// ---- XTS/Mover/types/ST_GEAR_DATA.TcDUT
{attribute 'pack_mode' := '2'}
TYPE ST_GEAR_DATA :
STRUCT
  rDeltaToMasterPos       : LREAL := 100.0;
  rModuloSyncPosSlave     : LREAL := 225.0;
  rMasterStartDistance    : LREAL :=   0.0;
  rGearNumerator          : LREAL :=   1.0;
  iGearDenumerator        : USINT :=   1;
END_STRUCT
END_TYPE

// ---- XTS/XtsStation/_types/ST_STATION_PARAMETER.TcDUT
TYPE ST_STATION_PARAMETER :
STRUCT
  sText             : STRING(80); // only description
  rPosWait          : REAL;       // start of station, a sending station is using this value to send mover to
  rReleaseDistance  : REAL;       // distance mover has to travel (from ActPos) in order for station to go back to mover detection

  rGap              : REAL;
  rVelo             : REAL;
  rAccDec           : REAL;
  rJerk             : REAL;

  // how many nests (stop positions) mover has to stop at (1 = default)
  nConfiguredStopCount  : USINT := 1; // 1-8 --> NestMask = BYTE

  // mover stop position in station, relative to rPosWait!!
  rPosStop          : ARRAY[1..8] OF LREAL;
END_STRUCT
END_TYPE

// ---- XTS/Xpu/types/ST_XPU_CTRL.TcDUT
{attribute 'pack_mode' := '2'}
TYPE ST_XPU_CTRL :
STRUCT
  Cmd             : E_XPU_CTRL;
END_STRUCT
END_TYPE

// ---- APPLICATION/GVL_APPLICATION.TcGVL
VAR_GLOBAL CONSTANT
  MAX_PROCESS       : UINT := 3;
END_VAR
{attribute 'qualified_only'}
VAR_GLOBAL
  MasterAxis              : Tc2_MC2.AXIS_REF;

  MasterPower             : Tc2_MC2.MC_Power;
  MasterReset             : Tc2_MC2.MC_Reset;
  MasterHalt              : Tc2_MC2.MC_Halt;
  MasterMoveVelo          : Tc2_MC2.MC_MoveVelocity;

  MoveData                : ST_MOVE_DATA;    // dynamic constraints for move commands
  GearData                : ST_GEAR_DATA;    // dynamic constraints and positions for GearIn/GearInPosCa

END_VAR

// ---- MSG/GVL_MSG.TcGVL
{attribute 'qualified_only'}
VAR_GLOBAL CONSTANT
  //-----------------------------------------------------------------------------
  // file paths for message system
  //  - compiler define option WIN switches to Windows file paths
  //-----------------------------------------------------------------------------
{IF defined (WIN)}
  {info 'WIN folders'}
  LOG_DIR               : STRING  := 'C:\TwinCAT\#MsgFiles\';
  CONFIG_DIR            : STRING  := 'C:\TwinCAT\XPU_PLC_StationConfig\';
{ELSE}
  {info 'BSD folders'}
  LOG_DIR               : STRING  := '/usr/local/etc/TwinCAT/#MsgFiles/';
  CONFIG_DIR            : STRING  := '/usr/local/etc/TwinCAT/XPU_PLC_StationConfig/';
{END_IF}

  LOG_FILE              : STRING  := 'MSG_XtsTransport_';
  CONFIG_FILE           : STRING  := 'Config_XPU_'; // OTCID of fb_Environment is added to name on writing

  MAX_MESSAGE           : UINT    := 200; // max entry in message list
END_VAR
VAR_GLOBAL
  Messages                        : ARRAY[1..MAX_MESSAGE] OF ST_Message;
  MessageIndex                    : UINT := 0; // message index
  MessageError                    : UINT := 0; // error counter

  fbLocalTime                     : fb_LocalTime;
  dtLocalTime                     : DT;
  sLocalTime                      : STRING;

  MessageLevelXpu                 : E_MessageType;
  MessageLevelStations            : ARRAY[1..MAX_STATION] OF E_MessageType;
  MessageLevelMovers              : ARRAY[1..MAX_MOVER]   OF E_MessageType;

  MessageLevelProcess             : ARRAY[1..MAX_PROCESS] OF E_MessageType;

{IF defined (TEST)}
  {info 'TEST logging enabled'}
  MessageLevel                    : E_MessageType := eMessageVerbose; // a lot of messages
{ELSE}
  MessageLevel                    : E_MessageType := eMessageError;    // not as much messages 
{END_IF}

END_VAR

// ---- XTS/GVL_XTS.TcGVL
{attribute 'qualified_only'}
VAR_GLOBAL
  //---------------------------------------------------------------------------
  // XTS Station
  //  - handshakes mover in station with extern control
  //  - station parameters (positions, gap, dyn. constraints, description...)
  StationStart        : ST_STATION_PARAMETER;   // Xts transport is sending all mover to this position (CMD_TRANSPORT_START)
  StationStartIndex   : UINT := 1;              // index of XtsStation where all movers are entered into linked list.

  // station handshaking with mover and extern process
  // station sends mover to target station/WaitPos
  // station adds mover data to LinkedList.AddTail() of target station
  Station             : ARRAY[1..MAX_STATION] OF fb_Station;
  StationList         : ARRAY[1..MAX_STATION] OF fb_Station_LinkedListCtrl;

  StationQueue        : ARRAY[1..MAX_STATION]    OF 
                        ARRAY[1..MAX_LIST_NODES] OF ST_STATION_MOVER_DATA;

  // interface for access to List methods
  StationListItf      : ARRAY[1..MAX_STATION] OF I_Station_LinkedList;

  // interface for access to station methods
  StationCtrlItf      : ARRAY[1..MAX_STATION] OF I_XtsTransport_Station;

  // ctrl / state datafields for extern control
  StationCtrl         : ARRAY[1..MAX_STATION] OF ST_STATION_CTRL;   // control for extern to write
  StationState        : ARRAY[1..MAX_STATION] OF ST_STATION_STATE;  // state for extern to read

  // station parameter
  StationParameter    : ARRAY[1..MAX_STATION] OF ST_STATION_PARAMETER; // XtsStation (fb_Station) positions and dyn constraints

  // static position offsets in stations
  PositionOffset      : ARRAY[1..MAX_STATION] OF T_NEST_OFFSET; // added to PosStop[] in XtsStation


  //---------------------------------------------------------------------------
  // XTS
  // XTS TransportUnit
  //  - handles request for XPU, Group, Mover, StartUp, ReStart
  XtsTransport        : fb_TransportUnit;         // manages members of XTS transport for extern to access

  XtsTransportCtrl    : ST_XTS_TRANSPORT_CTRL;    // control of XTS transport for extern to write
  XtsTransportState   : ST_XTS_TRANSPORT_STATE;   // state   of XTS transport for extern to read


  //---------------------------------------------------------------------------
  // XPU
  // XTS-Utility checks
  // XTS-Utility interfaces for you to use
  Xpu             : fb_XpuCtrl;

  XpuCtrl         : ST_XPU_CTRL;
  XpuState        : ST_XPU_STATE;
  XpuInfo         : ST_XPU_INFO;
  XpuModules      : ARRAY[1..MAX_MODULE] OF Tc3_XTS_Utility.ST_InfoDataView;


  //---------------------------------------------------------------------------
  // Collision avoidance group CA
  //
  // - add mover to group
  // - build group
  // - clear group
  CaGroup         : FB_CaGroup;                   // cyclic check of CaGroup state and errors; carries methods for handling CaGroup
  CaGroupItf      : I_XtsTransport_CaGroup;       // Interface used by fb_TransportUnit

  // cyclic mapping to MOTION/Objects/CaGroup 
  CaGroupRef      : Tc3_McCoordinatedMotion.AXES_GROUP_REF;

  // Info data from CaGroup FB
  CaGroupInfo     : ST_GROUP_INFO;                // cyclic info about CaGroup for fb_TransportUnit to read
  //---------------------------------------------------------------------------

  //---------------------------------------------------------------------------
  // MC2 encapsulation, CA movement
  Mover           : ARRAY[1..MAX_MOVER] OF fb_MoverCtrl;    // MC and CA methods for mover; cyclic check for individual command on mover

  MoverCtrl       : ARRAY[1..MAX_MOVER] OF ST_MOVER_CTRL;   // control of individual mover for extern to write
  MoverState      : ARRAY[1..MAX_MOVER] OF ST_MOVER_STATE;  // state   of individual mover for extern to read

  MoverItf        : ARRAY[1..MAX_MOVER] OF I_XtsTransport_Mover;  // Interface used by fb_TransportUnit

  LastPosition    : ARRAY[1..MAX_MOVER] OF LREAL;           // on execute of any movement, value is saved here (used by fb_Mover)
  LastGap         : ARRAY[1..MAX_MOVER] OF LREAL;           // on execute of any movement, value is saved here (used by fb_Mover)

  MoverInfo       : ARRAY[1..MAX_MOVER] OF ST_MOVER_INFO;   // cyclic info about mover for extern to read

  MoveData        : ARRAY[1..MAX_MOVER] OF ST_MOVE_DATA;    // dynamic constraints for move commands
  GearData        : ARRAY[1..MAX_MOVER] OF ST_GEAR_DATA;    // dynamic constraints and positions for GearIn/GearInPosCa
  
  // cyclic mapping to MOTION/Axes
  AxisRefMover    : ARRAY[1..MAX_MOVER] OF Tc2_MC2.AXIS_REF;
  //---------------------------------------------------------------------------
END_VAR

// ---- XTS/XTS_Parameter.TcGVL
//{attribute 'qualified_only'}
VAR_GLOBAL CONSTANT
// HAUD 2025 08 09
//
//    XTS_TRANSPORT_LAYER project
//    
//    MIT License
//    
//    Copyright (c) 2025 HAUD
//    
//    Permission is hereby granted, free of charge, to any person obtaining a copy
//    of this software and associated documentation files (the "Software"), to deal
//    in the Software without restriction, including without limitation the rights
//    to use, copy, modify, merge, publish, distribute, sublicense, and/or sell
//    copies of the Software, and to permit persons to whom the Software is
//    furnished to do so, subject to the following conditions:
//    
//    The above copyright notice and this permission notice shall be included in all
//    copies or substantial portions of the Software.
//    
//    THE SOFTWARE IS PROVIDED "AS IS", WITHOUT WARRANTY OF ANY KIND, EXPRESS OR
//    IMPLIED, INCLUDING BUT NOT LIMITED TO THE WARRANTIES OF MERCHANTABILITY,
//    FITNESS FOR A PARTICULAR PURPOSE AND NONINFRINGEMENT. IN NO EVENT SHALL THE
//    AUTHORS OR COPYRIGHT HOLDERS BE LIABLE FOR ANY CLAIM, DAMAGES OR OTHER
//    LIABILITY, WHETHER IN AN ACTION OF CONTRACT, TORT OR OTHERWISE, ARISING FROM,
//    OUT OF OR IN CONNECTION WITH THE SOFTWARE OR THE USE OR OTHER DEALINGS IN THE
//    SOFTWARE.

  Version             : STRING  := '4.00.11';

  MAX_MOVER           : UINT    := TO_UINT(Tc3_XTS_Utility.TcIoXtsEnvironmentParameterList.MaxXtsMoversPerXpu);
  MAX_MODULE          : UINT    := TO_UINT(Tc3_XTS_Utility.TcIoXtsEnvironmentParameterList.MaxModulesPerPart);
  MAX_PART            : UINT    := TO_UINT(Tc3_XTS_Utility.TcIoXtsEnvironmentParameterList.MaxXtsPartsPerXpu);
  MAX_TRACK           : UINT    := TO_UINT(Tc3_XTS_Utility.TcIoXtsEnvironmentParameterList.MaxXtsTracksPerXpu);
  MAX_GROUP           : UINT    := TO_UINT(Tc3_XTS_Utility.TcIoXtsEnvironmentParameterList.MaxXtsCaGroup);

  MAX_INFO_SERVER     : UINT    := TO_UINT(Tc3_XTS_Utility.TcIoXtsEnvironmentParameterList.MaxXtsInfoServer);
  MAX_INFO_STATION    : UINT    := TO_UINT(Tc3_XTS_Utility.TcIoXtsEnvironmentParameterList.MaxXtsInfoStation);
  MAX_INFO_STOP_POS   : UINT    := TO_UINT(Tc3_XTS_Utility.TcIoXtsEnvironmentParameterList.MaxXtsStopPositionsPerStation);

  MAX_PARAMETER_SET   : UINT    := TO_UINT(Tc3_XTS_Utility.TcIoXtsEnvironmentParameterList.MaxXtsParameterSet);

  MAX_NCT_BASE_UNIT   : UINT    := TO_UINT(Tc3_XTS_Utility.TcIoXtsEnvironmentParameterList.MaxXtsNctBaseUnitInterfaces);

  MAX_STATION         : UINT    := 2;

  MAX_STATION_NEST    : UINT    := TO_UINT(SIZEOF(ST_STATION_STATE.nMask)*8);
  // MAX_LIST_NODES      : UINT    := MAX_MOVER;
  MAX_LIST_NODES      : UINT    := 24; // visualization can not handle access to MAX_MOVER
  MAX_MASTER          : UINT    := 1;
END_VAR

// ---- XTS/Mover/I_XtsTransport_Mover.TcIO
INTERFACE I_XtsTransport_Mover

METHOD Disable : E_PROGRESS
VAR_INPUT
  Execute             : BOOL;
END_VAR
END_METHOD

METHOD Enable : E_PROGRESS
VAR_INPUT
  Execute             : BOOL;
END_VAR
END_METHOD

METHOD GearIn : E_PROGRESS;
VAR_INPUT
  Execute             : BOOL;
  stMoveData          : ST_MOVE_DATA;
  stGearData          : ST_GEAR_DATA;
END_VAR
END_METHOD

METHOD GearInPosCa : E_PROGRESS
VAR_INPUT
  Execute             : BOOL;
  stMoveData          : ST_MOVE_DATA;
  stGearData          : ST_GEAR_DATA;  
END_VAR
END_METHOD

METHOD GearOut : E_PROGRESS
VAR_INPUT
  Execute             : BOOL;
END_VAR
END_METHOD

METHOD Halt : E_PROGRESS
VAR_INPUT
  Execute             : BOOL;
  stMoveData          : ST_MOVE_DATA;
END_VAR
END_METHOD

METHOD HaltCa : E_PROGRESS
VAR_INPUT
  Execute             : BOOL;
  stMoveData          : ST_MOVE_DATA;
END_VAR
END_METHOD

PROPERTY MessageLevel : e_messagetype
SET
END_SET
END_PROPERTY

PROPERTY ModuloTurn : dint
GET
END_GET
END_PROPERTY

METHOD MoveToPos : E_PROGRESS
VAR_INPUT
  Execute             : BOOL;
  stMoveData          : ST_MOVE_DATA;
END_VAR
END_METHOD

METHOD MoveToPosCa : E_PROGRESS
VAR_INPUT
  Execute             : BOOL;
  stMoveData          : ST_MOVE_DATA;
END_VAR
END_METHOD

PROPERTY RailLength : LREAL
GET
END_GET
SET
END_SET
END_PROPERTY

METHOD Reset : E_PROGRESS
VAR_INPUT
  Execute             : BOOL;
END_VAR
END_METHOD

METHOD SendToAbsPosCa : E_PROGRESS
VAR_INPUT
  Execute             : BOOL;
  stMoveData          : ST_MOVE_DATA;
END_VAR
END_METHOD

METHOD SendToModuloPosCa : E_PROGRESS
VAR_INPUT
  Execute             : BOOL;
  stMoveData          : ST_MOVE_DATA;
END_VAR
END_METHOD

METHOD Stop : E_PROGRESS
VAR_INPUT
  Execute             : BOOL;
  stMoveData          : ST_MOVE_DATA;
END_VAR
END_METHOD

END_INTERFACE

// ---- MAIN.TcPOU
//---------------------------------------------------------------------------------------------------------------
//
//  HAUD 2024.10.02
//
//  - XTS_DEMO_GEAR_IN_POS_CA
//
//  - XTS_TRANSPORT_LAYER
//  - transport layer members:
//    - CaGroup
//      - access to Group functions
//
//    - Mover
//      - access to MC and CA motion functions
//
//    - Xpu (ProcessingUnit)
//      - access to TcCOM Objects in Environment
//
//    - Transport Control Unit
//      - coordinates members to get XTS in defined states
//
//  - global datafields for mrmbers in GVL_XTS namespace
//  - global interface datafields for use in members
//  - structures are assigned by reference for every member
//
//---------------------------------------------------------------------------------------------------------------
// HAUD 2024 05 29
//
//    XTS_TRANSPORT_LAYER project
//    
//    MIT License
//    
//    Copyright (c) 2024 HAUD
//    
//    Permission is hereby granted, free of charge, to any person obtaining a copy
//    of this software and associated documentation files (the "Software"), to deal
//    in the Software without restriction, including without limitation the rights
//    to use, copy, modify, merge, publish, distribute, sublicense, and/or sell
//    copies of the Software, and to permit persons to whom the Software is
//    furnished to do so, subject to the following conditions:
//    
//    The above copyright notice and this permission notice shall be included in all
//    copies or substantial portions of the Software.
//    
//    THE SOFTWARE IS PROVIDED "AS IS", WITHOUT WARRANTY OF ANY KIND, EXPRESS OR
//    IMPLIED, INCLUDING BUT NOT LIMITED TO THE WARRANTIES OF MERCHANTABILITY,
//    FITNESS FOR A PARTICULAR PURPOSE AND NONINFRINGEMENT. IN NO EVENT SHALL THE
//    AUTHORS OR COPYRIGHT HOLDERS BE LIABLE FOR ANY CLAIM, DAMAGES OR OTHER
//    LIABILITY, WHETHER IN AN ACTION OF CONTRACT, TORT OR OTHERWISE, ARISING FROM,
//    OUT OF OR IN CONNECTION WITH THE SOFTWARE OR THE USE OR OTHER DEALINGS IN THE
//    SOFTWARE.
//---------------------------------------------------------------------------------------------------------------
PROGRAM MAIN
VAR
	bInit 				: BOOL;
  eInit         : E_PROGRESS;

  nStation,
	nMover,
  nMoverSelected,
  nStationSelected,
  nStationParameter   : UINT;

  sStationText        : STRING(30);

  eTransportState     : E_XTS_TRANSPORT_STATE;
  eTransportResult    : E_PROGRESS;

  eXpuState           : E_XPU_STATE;
  eXpuResult          : E_PROGRESS;
  eXpuCheck           : E_XPU_CHECK;

  eMoverState         : E_MOVER_STATE;
  eMoverResult        : E_PROGRESS;

  sCaGroupState,
  sTransportState,
  sTransportCheck,
  sTransportResult,
  sXpuState,
  sXpuResult,
  sXpuCheck,
  sXpuOpMode,
  sXpuMoverdetectionMode,
  sXpuMoverAssignement,
  sMoverState,
  sMoverResult,
  sStationState,
  sStationStateMask,
  sStationCtrlMask        : STRING;

  bStationEnable,
  bStationEnter,
  bStationStart,
  bStationDone,
  bStationOut,
  bStationGone            : BOOL;

  tStationSelectedQueue   : ARRAY[1..MAX_LIST_NODES] OF ST_STATION_MOVER_DATA;

  tonWriteLog             : Tc2_Standard.TON;
  tWriteLog               : TIME := T#5S;
END_VAR

//############################################################################
// Local time; used for timestamps
//############################################################################
GVL_MSG.fbLocalTime(
                    sLocalTime                => GVL_MSG.sLocalTime, 
                    dtLocalTime               => GVL_MSG.dtLocalTime);
//############################################################################

//############################################################################
// 	example for init sequence
//############################################################################	
IF NOT bInit
THEN
  CASE eInit
  OF
    E_PROGRESS.PROGRESS_INVALID,
    E_PROGRESS.PROGRESS_DONE:         // clear command interface
      eInit                                   := E_PROGRESS.PROGRESS_BUSY;
      GVL_XTS.XpuCtrl.Cmd                     := E_XPU_CTRL.XTS_CMD_NULL;
      GVL_MSG.MessageLevelXpu                 := GVL_MSG.MessageLevel;
      GVL_XTS.CaGroup.MessageLevel            := GVL_MSG.MessageLevel;
      FOR nStation := 1 TO MAX_STATION
      DO
        GVL_MSG.MessageLevelStations[nStation]:= GVL_MSG.MessageLevel;
      END_FOR
      FOR nMover := 1 TO MAX_MOVER
      DO
        GVL_MSG.MessageLevelMovers[nMover]    := GVL_MSG.MessageLevel;
      END_FOR


    E_PROGRESS.PROGRESS_BUSY:         // init Xpu, ProcessingUnit, MotorModules
      eInit                                   := E_PROGRESS.PROGRESS_PREPARE;
      GVL_XTS.XpuCtrl.Cmd                     := E_XPU_CTRL.XTS_CMD_INIT;

    E_PROGRESS.PROGRESS_PREPARE:      // wait for init to be done
      IF (GVL_XTS.XpuState.State      = E_XPU_STATE.XTS_INIT + E_PROGRESS.PROGRESS_DONE)
      THEN
        eInit                                 := E_PROGRESS.PROGRESS_STARTUP;
        GVL_XTS.XpuCtrl.Cmd                   := E_XPU_CTRL.XTS_IDLE;
      END_IF

    E_PROGRESS.PROGRESS_STARTUP:      // assign mover interfaces
      eInit                                   := E_PROGRESS.PROGRESS_CHECK;
      FOR nMover := 1 TO MAX_MOVER
      DO
        GVL_XTS.MoverItf[nMover]              := GVL_XTS.Mover[nMover];
      END_FOR

    E_PROGRESS.PROGRESS_CHECK:        // assign CaGroup interface
      eInit                                   := E_PROGRESS.PROGRESS_OCCUPIED;
      GVL_XTS.CaGroupItf                      := GVL_XTS.CaGroup;

    E_PROGRESS.PROGRESS_OCCUPIED:     // StartStation for XtsTransportCtrl.Cmd := E_XTS_TRANSPORT_CTRL.CMD_TRANSPORT_START;
      eInit                                   := E_PROGRESS.PROGRESS_WORKING;
      // where to start?
      GVL_XTS.XtsTransport.StationStartIndex  := 0; // no stations in use in this example, therefore no StartStation

      // IF you use stations, initialize them here, before StationStart is initialized!

    E_PROGRESS.PROGRESS_WORKING:
      // Start Position parameters
      GVL_XTS.StationStart.rPosWait           :=     10.0; // this value may differ from the GVL_XTS.StationParameter[StartStationIndex], IF it differs, you MUST have room for positive movement to GVL_XTS.StationParameter[StartStationIndex].rWaitPos
      GVL_XTS.StationStart.rGap               :=    250.0; // may differ, or just copy from GVL_XTS.StationParameter[StartStationIndex]
      GVL_XTS.StationStart.rVelo              :=    750.0; // may differ, or just copy from GVL_XTS.StationParameter[StartStationIndex]
      GVL_XTS.StationStart.rAccDec            :=  12000.0; // may differ, or just copy from GVL_XTS.StationParameter[StartStationIndex]
      GVL_XTS.StationStart.rJerk              := 400000.0; // may differ, or just copy from GVL_XTS.StationParameter[StartStationIndex], the movements are more robust if you keep this value in a narrow range, since jumps lead to adjusting movements within the CA Group

      IF (GVL_XTS.XtsTransport.StationStartIndex > 0) AND
         (GVL_XTS.XtsTransport.StationStartIndex < MAX_STATION+1)
      THEN
        GVL_XTS.StationStart.nConfiguredStopCount := GVL_XTS.StationParameter[GVL_XTS.XtsTransport.StationStartIndex].nConfiguredStopCount;
      END_IF

      bInit                                           := TRUE;
      eInit                                           := E_PROGRESS.PROGRESS_DONE;
  END_CASE
END_IF

//############################################################################
// 	XTS Transport Unit
//############################################################################
//  - main control function block for transport layer
//  - requires access to member controls
//    - Xpu
//    - CaGroup
//    - Mover
//    - Station Control
//    - Station LinkedList Interface
//############################################################################
//
// cyclic call
GVL_XTS.XtsTransport();

// main control
GVL_XTS.XtsTransport.Ctrl               REF= GVL_XTS.XtsTransportCtrl;   // main control
GVL_XTS.XtsTransport.State              REF= GVL_XTS.XtsTransportState;  // main state
                                        
// member controls                      
GVL_XTS.XtsTransport.XpuCtrl            REF= GVL_XTS.XpuCtrl;
GVL_XTS.XtsTransport.XpuState           REF= GVL_XTS.XpuState;
GVL_XTS.XtsTransport.XpuInfo            REF= GVL_XTS.XpuInfo;
                                        
GVL_XTS.XtsTransport.GroupItf           :=   GVL_XTS.CaGroupItf;
GVL_XTS.XtsTransport.GroupInfo          REF= GVL_XTS.CaGroupInfo;
                                        
GVL_XTS.XtsTransport.MoverItf           REF= GVL_XTS.MoverItf;
GVL_XTS.XtsTransport.MoverInfo          REF= GVL_XTS.MoverInfo;
GVL_XTS.XtsTransport.MoverLastPosition  REF= GVL_XTS.LastPosition;
GVL_XTS.XtsTransport.MoverLastGap       REF= GVL_XTS.LastGap;
                                        
GVL_XTS.XtsTransport.StationStart       REF= GVL_XTS.StationStart;      // start position for E_XTS_TRANSPORT_CTRL.CMD_TRANSPORT_START
GVL_XTS.XtsTransport.StationCtrlItf     REF= GVL_XTS.StationCtrlItf;    // station interfaces are required for accessing station methods
GVL_XTS.XtsTransport.StationListsItf    REF= GVL_XTS.StationListItf;    // list interface is required for access to linked list methods
GVL_XTS.XtsTransport.StationControl     REF= GVL_XTS.StationCtrl;
GVL_XTS.XtsTransport.StationState       REF= GVL_XTS.StationState;
//############################################################################



//############################################################################
// 	XTS Stations
//############################################################################	
FOR nStation := 1 TO MAX_STATION
DO
  GVL_XTS.Station[nStation].StationId   := nStation;
  GVL_XTS.Station[nStation].MessageLevel:= GVL_MSG.MessageLevelStations[nStation];

  GVL_XTS.StationListItf[nStation]      := GVL_XTS.StationList[nStation];   // interfaces for list methods
  GVL_XTS.StationCtrlItf[nStation]      := GVL_XTS.Station[nStation];       // interfaces for station methods

  GVL_XTS.Station[nStation].Ctrl        REF= GVL_XTS.StationCtrl;           // station ctrl from extern
  GVL_XTS.Station[nStation].State       REF= GVL_XTS.StationState;          // station state to extern

  GVL_XTS.Station[nStation].ItfStations REF= GVL_XTS.StationListItf;        // give every station all list interfaces for writing mover tickets
  GVL_XTS.Station[nStation].ItfMover    REF= GVL_XTS.MoverItf;              // give every station all mover interfaces for movement in / out of station
  GVL_XTS.Station[nStation].Mover       REF= GVL_XTS.AxisRefMover;          // AXIS_REF to read infos from
  GVL_XTS.Station[nStation].MoverOffset REF= GVL_XTS.PositionOffset;        // static offsets for all stations, all movers, all stop positions


  GVL_XTS.Station[nStation].StationParameter  REF= GVL_XTS.StationParameter;// give every station all station parameters for sending to WaitPos of target station

  // cyclic call
  GVL_XTS.Station[nStation].Cycle();                                        // cycle for handshaking with extern

  // Queue data for each station
  GVL_XTS.StationQueue[nStation]        := GVL_XTS.StationListItf[nStation].Data;
END_FOR
//############################################################################



//############################################################################
// 	XPU environment
//############################################################################	
GVL_XTS.Xpu.XpuInstance               :=   1;
GVL_XTS.Xpu.MessageLevel              :=   GVL_MSG.MessageLevelXpu;

GVL_XTS.Xpu.Ctrl                      REF= GVL_XTS.XpuCtrl;
GVL_XTS.Xpu.State                     REF= GVL_XTS.XpuState;
GVL_XTS.Xpu.XpuModuleInfoData         REF= GVL_XTS.XpuModules;

GVL_XTS.Xpu.CaGroupOID                :=   GVL_XTS.CaGroup.GroupInfo.CaGroupOID;

// cyclic call
GVL_XTS.Xpu();
GVL_XTS.XpuInfo                       :=   GVL_XTS.Xpu.XpuInfo;
//############################################################################


//############################################################################	
// 	CA-Group Class
//############################################################################	
// assignment
GVL_XTS.CaGroup.AxisRef               REF= GVL_XTS.AxisRefMover;
// Interface to Mover methods
GVL_XTS.CaGroup.MoverItf              REF= GVL_XTS.MoverItf; 

GVL_XTS.CaGroup.GroupRef              REF= GVL_XTS.CaGroupRef;

// cyclic call
GVL_XTS.CaGroup.InfoCycle(TRUE); // read group status

// InfoData from group
GVL_XTS.CaGroupInfo                   :=   GVL_XTS.CaGroup.GroupInfo;

// Interface of CaGroup
GVL_XTS.CaGroupItf                    :=   GVL_XTS.CaGroup;
//############################################################################


//############################################################################
// Mover Class	
//############################################################################	
FOR nMover := 1 TO MAX_MOVER
DO
  GVL_XTS.Mover[nMover].MoverId       :=   nMover;
  GVL_XTS.Mover[nMover].RailLength    :=   GVL_XTS.Xpu.RailLength;  // mover needs RailLength, in order to calc absolute position from modulo input
  GVL_XTS.Mover[nMover].MessageLevel  :=   GVL_MSG.MessageLevelMovers[nMover];

  GVL_XTS.Mover[nMover].Ctrl          REF= GVL_XTS.MoverCtrl;       // mover control from extern
  GVL_XTS.Mover[nMover].State         REF= GVL_XTS.MoverState;      // mover state to extern

  GVL_XTS.Mover[nMover].MoveData      REF= GVL_XTS.MoveData;        // dyn constraints for extern to write
  GVL_XTS.Mover[nMover].GearData      REF= GVL_XTS.GearData;        // GearIn/GearInPosCa data fro extern to write

  // assignment	
  GVL_XTS.Mover[nMover].Mover         REF= GVL_XTS.AxisRefMover[nMover];  // axis reference to Mover function block
  GVL_XTS.Mover[nMover].LastGap       REF= GVL_XTS.LastGap[nMover];       // reference to last used gap value datafield
  GVL_XTS.Mover[nMover].LastPosition  REF= GVL_XTS.LastPosition[nMover];  // reference to last position datafield

  GVL_XTS.Mover[nMover].MoverInfo		  REF= GVL_XTS.MoverInfo[nMover];     // refernence to mover info data (ActPos, SetPos, ...)

  GVL_XTS.MoverItf[nMover]            :=   GVL_XTS.Mover[nMover];

  // master axis assigned to mover
  GVL_XTS.Mover[nMover].Master        REF= GVL_APPLICATION.MasterAxis;    // GearInPosCa conveyer axis is master in this example

  // cyclic call
  GVL_XTS.Mover[nMover].Cycle();  // call AXIS_REF()
  GVL_XTS.Mover[nMover]();        // call Ctrl/State
END_FOR


//############################################################################


//############################################################################
// /logging
//############################################################################
tonWriteLog(IN:= TRUE, PT := tWriteLog);

IF (tonWriteLog.Q)
THEN
  MessageData.bWriteFile      := TRUE;
  tonWriteLog(IN:= FALSE);
END_IF

//-----------------------------------------------------------------------------------------------------------------
// write message list to file
//-----------------------------------------------------------------------------------------------------------------
MessageData(pList			        := ADR(GVL_MSG.Messages),
			      pLocalTime        := ADR(GVL_MSG.dtLocalTime), 
			      bBusy=> );

// clear write trigger
IF MessageData.bWriteFile AND
   MessageData.bDone
THEN
  MessageData.bWriteFile      := FALSE;
END_IF
//############################################################################
// logging/
//############################################################################



//############################################################################
// Visualization data	
//############################################################################	
// get enumerations from XPU for visu:
eTransportState                       := f_GetState   (GVL_XTS.XtsTransportState.State);
eTransportResult                      := f_GetProgress(GVL_XTS.XtsTransportState.State);

eXpuState                             := f_GetState   (GVL_XTS.XpuState.State);
eXpuResult                            := f_GetProgress(GVL_XTS.XpuState.State);

eXpuCheck                             := GVL_XTS.XpuState.Check;

// display xpu state and result in visu
// get strings and info
sCaGroupState                         := TO_STRING(GVL_XTS.CaGroupInfo.CaGroupState);

sTransportState                       := TO_STRING(eTransportState);
sTransportCheck                       := TO_STRING(GVL_XTS.XtsTransportState.Check);
sTransportResult                      := TO_STRING(eTransportResult);

sXpuState                             := TO_STRING(eXpuState);
sXpuResult                            := TO_STRING(eXpuResult);
sXpuCheck                             := TO_STRING(eXpuCheck);

sXpuOpMode                            := GVL_XTS.Xpu.OpModeToString();
sXpuMoverdetectionMode                := GVL_XTS.Xpu.IdDetectionModeToString();
sXpuMoverAssignement                  := GVL_XTS.Xpu.MoverPositionAssignementToString();

nMoverSelected                        := SEL((nMoverSelected<1), nMoverSelected, 1);
nMoverSelected                        := SEL((nMoverSelected>MAX_MOVER), nMoverSelected, MAX_MOVER);

nStationSelected                      := SEL((nStationSelected<1), nStationSelected, 1);
nStationSelected                      := SEL((nStationSelected>MAX_STATION), nStationSelected, MAX_STATION);

bStationEnable                        := SEL((GVL_XTS.StationCtrl[nStationSelected].eCmd = E_STATION_CTRL.STATION_ENABLE),        FALSE, TRUE);
bStationEnter                         := SEL((GVL_XTS.StationCtrl[nStationSelected].eCmd = E_STATION_CTRL.STATION_MOVER_ENTER),   FALSE, TRUE);
bStationStart                         := SEL((GVL_XTS.StationCtrl[nStationSelected].eCmd = E_STATION_CTRL.STATION_PROCESS_START), FALSE, TRUE);
bStationDone                          := SEL((GVL_XTS.StationCtrl[nStationSelected].eCmd = E_STATION_CTRL.STATION_PROCESS_DONE),  FALSE, TRUE);
bStationOut                           := SEL((GVL_XTS.StationCtrl[nStationSelected].eCmd = E_STATION_CTRL.STATION_MOVER_OUT),     FALSE, TRUE);
bStationGone                          := SEL((GVL_XTS.StationCtrl[nStationSelected].eCmd = E_STATION_CTRL.STATION_MOVER_GONE),    FALSE, TRUE);

eMoverState                           := f_GetState   (GVL_XTS.MoverState[nMoverSelected].State);
eMoverResult                          := f_GetProgress(GVL_XTS.MoverState[nMoverSelected].State);

sMoverState                           := TO_STRING(eMoverState);
sMoverResult                          := TO_STRING(eMoverResult);

sStationState                         := TO_STRING(GVL_XTS.StationState[nStationSelected].eState);
sStationStateMask                     := Tc2_Utilities.BYTE_TO_BINSTR(GVL_XTS.StationState[nStationSelected].nMask, 8);
sStationCtrlMask                      := Tc2_Utilities.BYTE_TO_BINSTR(GVL_XTS.StationCtrl[nStationSelected].nMask, 8);

tStationSelectedQueue                 := GVL_XTS.StationQueue[nStationSelected];

END_PROGRAM

// ---- MSG/MessageData.TcPOU
PROGRAM MessageData
VAR CONSTANT
{attribute 'hide'}
  STR_LEN       : UDINT := 131_070;
END_VAR
VAR_INPUT
	bPowerFail		: BOOL;   // UPS switch
	bWriteFile		: BOOL;   // manual write of list
	bReset				: BOOL;
	pList					: POINTER TO ARRAY[1..GVL_MSG.MAX_MESSAGE] OF ST_Message; // attach your list here
	pLocalTime		: POINTER TO DT; 
END_VAR
VAR_OUTPUT
	bBusy					: BOOL;
  bDone         : BOOL;
	VisuList		  : ARRAY[1..GVL_MSG.MAX_MESSAGE] OF ST_Message;
END_VAR
VAR
	eState 				: E_MESSAGE_STATE;

	rtrigReset		: Tc2_Standard.R_TRIG;
	aWriteList		: ARRAY[1..GVL_MSG.MAX_MESSAGE] OF ST_Message;
	sWriteData		: STRING(STR_LEN);
	sNewLine			: STRING := '$N';
	sTab					: STRING := '$T';
	iCount, 
	iStart, 
	iEnd					: UINT;

	fbCreateDir		: Tc2_System.FB_CreateDir;
	sTmp          : STRING(256);
	sFilename			: STRING(256);
	sFolderDate		: STRING;
	bFileCreated	: BOOL;

	fbFileOpen		  : Tc2_System.FB_FileOpen;
	fbFileWrite		  : Tc2_System.FB_FileWrite;
	fbFileClose		  : Tc2_System.FB_FileClose;

  ivis          : UINT;

  bBusyWrite,
  bErrorWrite   : BOOL;
  nErrorWrite   : UDINT;
  nStateWrite   : UINT;
END_VAR

//-----------------------------------------------------------------------------
// check pointers
//-----------------------------------------------------------------------------
IF NOT (pList <> 0) OR
   NOT (pLocalTime <> 0)
THEN
  eState                      := MSG_INVALID_POINTERS;
  RETURN;
END_IF
//-----------------------------------------------------------------------------
// check date
// new message file for a new day
//-----------------------------------------------------------------------------
IF (FolderDate(pLocalTime) <> sFolderDate)
THEN
  bFileCreated                := FALSE;
END_IF
//-----------------------------------------------------------------------------
//----------------------------------------------------------------------------- 
rtrigReset(CLK:= bReset);
IF rtrigReset.Q
THEN
  bReset                      := FALSE;
  eState                      := MSG_NULL;
END_IF
//-----------------------------------------------------------------------------
//-----------------------------------------------------------------------------
CASE eState OF
  MSG_NULL:
    bBusy                     := 
    bDone                     := FALSE;

    IF (GVL_MSG.MessageIndex > GVL_MSG.MAX_MESSAGE/2)
    THEN
      eState                  := MSG_INIT;

    ELSIF (bWriteFile) OR (bPowerFail)
    THEN
      eState                  := MSG_INIT;

      IF (GVL_MSG.MessageIndex = 0)
      THEN
        bBusy                 := TRUE;
        eState                := MSG_WRITE_FILE_DONE;
      END_IF
    END_IF
END_CASE
//-----------------------------------------------------------------------------
CASE eState OF
  MSG_INIT:
    WriteData(FALSE);

    // clear intern list
    memset(ADR(aWriteList),     0, SIZEOF(aWriteList));

    // copy from attached list to local
    memcpy(ADR(aWriteList), pList, SIZEOF(aWriteList));

    // clear attached list
    memset(pList, 0, SIZEOF(aWriteList));

    bBusy                     := TRUE;
    iStart 	                  := 1;
    iEnd 		                  := SEL((GVL_MSG.MessageIndex > GVL_MSG.MAX_MESSAGE-1),
                                      GVL_MSG.MessageIndex,
                                      GVL_MSG.MAX_MESSAGE);
    GVL_MSG.MessageIndex      := 0;

    IF NOT bFileCreated
    THEN
      // folder and filename have to be created
      eState                  := MSG_ROOT;
    ELSE
      // folder and file already exist
      eState                  := MSG_LINE_START;
    END_IF
END_CASE
//-----------------------------------------------------------------------------
CASE eState OF
  MSG_ROOT:
    eState                    := MSG_ROOT_CREATE;
    fbCreateDir.sPathName     := left(GVL_MSG.LOG_DIR,len(GVL_MSG.LOG_DIR)-1);
    fbCreateDir(
            bExecute	        := FALSE);
  
  MSG_ROOT_CREATE:
    (* create root folder *)
    fbCreateDir(
            bExecute	        := TRUE);
    IF fbCreateDir.bBusy
    THEN
      eState                  := MSG_ROOT_CREATE_BUSY;
    END_IF
  
  MSG_ROOT_CREATE_BUSY:
    fbCreateDir(
            bExecute	        := TRUE);
    IF NOT fbCreateDir.bBusy
    THEN
      eState                  := MSG_FOLDER;
    END_IF
  
  MSG_FOLDER:
    eState                    := MSG_FOLDER_CREATE;
    sFolderDate               := FolderDate(pLocalTime);
    fbCreateDir.sPathName     := concat(GVL_MSG.LOG_DIR, sFolderDate);
    fbCreateDir(
            bExecute	        := FALSE);

  MSG_FOLDER_CREATE:
    (* create active folder *)
    fbCreateDir(
            bExecute	        := TRUE);
    IF fbCreateDir.bBusy
    THEN
      eState                  := MSG_FOLDER_CREATE_BUSY;
    END_IF
  
  MSG_FOLDER_CREATE_BUSY:
    fbCreateDir(
            bExecute	        := TRUE);
    IF NOT fbCreateDir.bBusy
    THEN
      eState                  := MSG_FILE_CREATE_DONE;
      fbCreateDir(
              bExecute	      := FALSE);
    END_IF
END_CASE
//-----------------------------------------------------------------------------
CASE eState OF
  MSG_FILE_CREATE_DONE:
    eState                    := MSG_LINE_START;
    bFileCreated              := TRUE;
    // build complete file path
    sTmp                      := concat(concat(GVL_MSG.LOG_FILE, sFolderDate),'.txt');
    sTmp                      := concat('\', sTmp);
    sFilename                 := concat(fbCreateDir.sPathName, sTmp);
END_CASE
//-----------------------------------------------------------------------------
CASE eState OF
  MSG_LINE_START:
    GVL_MSG.MessageError      := 0;
    eState                    := MSG_LINE_BUILD;
    iCount                    := iStart;
    memset(ADR(sWriteData),0,SIZEOF(sWriteData));
END_CASE
//-----------------------------------------------------------------------------
CASE eState OF
  MSG_LINE_BUILD:
    eState                    := MSG_LINE_CHECK;
    IF (aWriteList[iCount].eType > E_MessageType.eMessageEmpty)
    THEN
      sTmp                    := TO_STRING(aWriteList[iCount].eType);
      sTmp                    := Tc2_Standard.CONCAT(sTmp, sTab);
      sTmp                    := Tc2_Standard.CONCAT(sTmp, aWriteList[iCount].tTime);
      sTmp                    := Tc2_Standard.CONCAT(sTmp, sTab);
      sTmp                    := Tc2_Standard.CONCAT(sTmp, Device_To_String(aWriteList[iCount].eDevice));
      sTmp                    := Tc2_Standard.CONCAT(sTmp, sTab);
      sTmp                    := Tc2_Standard.CONCAT(sTmp, TO_STRING(aWriteList[iCount].eSubdevice));
      sTmp                    := Tc2_Standard.CONCAT(sTmp, sTab);
      sTmp                    := Tc2_Standard.CONCAT(sTmp, TO_STRING(aWriteList[iCount].iErrorNumber));
      sTmp                    := Tc2_Standard.CONCAT(sTmp, sTab);
      sTmp                    := Tc2_Standard.CONCAT(sTmp, aWriteList[iCount].sText);
      sTmp                    := Tc2_Standard.CONCAT(sTmp, sNewLine);
      Builder(ADR(sTmp), ADR(sWriteData), StringLen(ADR(sTmp)));
    END_IF
    iCount                    := iCount + 1;
END_CASE
//-----------------------------------------------------------------------------
CASE eState OF
  MSG_LINE_CHECK:
  IF NOT (iCount > iEnd)
  THEN
    eState                    := MSG_LINE_BUILD;
  ELSE
    IF (StringLen(ADR(sWriteData)) > 1)
    THEN
      eState                  := MSG_WRITE_FILE_BUSY;
    ELSE
      eState                  := MSG_WRITE_FILE_DONE;
    END_IF
  END_IF
  
  MSG_WRITE_FILE_BUSY:
  IF WriteData(TRUE)
  THEN
    eState                    := MSG_WRITE_FILE_END;
  END_IF
  
  MSG_WRITE_FILE_END:
  WriteData(FALSE);
  eState                      := MSG_WRITE_FILE_DONE;
  
  MSG_WRITE_FILE_DONE:
  bDone                       := TRUE;
  IF NOT (bWriteFile)
  THEN
    eState                    := MSG_NULL;
  END_IF
END_CASE
//-----------------------------------------------------------------------------
//-----------------------------------------------------------------------------
// visu message list
//-----------------------------------------------------------------------------
memset(ADR(VisuList),0,SIZEOF(VisuList));
// copy last written message list to visu message list
memcpy(ADR(VisuList), ADR(aWriteList), SIZEOF(VisuList));
//-----------------------------------------------------------------------------

METHOD Builder : BOOL // string concat for length > 255
VAR_INPUT
  pInString   : POINTER TO STRING;
  pOutString  : POINTER TO STRING(STR_LEN);
  Length      : UINT;
END_VAR
VAR
  Counter     : UDINT;
  pInWork     : POINTER TO BYTE;
  pOutWork    : POINTER TO BYTE;
END_VAR
pOutWork := pOutString;
pInWork := pInString;
Counter := 0;

(*check termination*)
WHILE (pOutWork^ <> 0) AND
      (Counter < STR_LEN+1)
DO
  Counter := Counter + 1;
  pOutWork := pOutWork + 1;
END_WHILE

(* append only if data fits into output *)
IF (Counter + Length < STR_LEN+1)
THEN

  (* append data *)
  FOR Counter := 1 TO Length
  DO
    pOutWork^ := pInWork^;
    pOutWork := pOutWork + 1;
    pInWork := pInWork + 1;
  END_FOR

  (* terminate *)
  pOutWork := pOutWork + 1;
  pOutWork^ := 0;
END_IF
END_METHOD

METHOD Device_to_String : string
VAR_INPUT
  eMsgDevice    : e_Device;
END_VAR
VAR
  sId                 : STRING := '_ID_';
  nId                 : UDINT;
END_VAR
IF (eMsgDevice < e_device.General)
THEN
  // below general case
  nId := TO_UDINT(eMsgDevice);
  sId := concat(sId, TO_STRING(nId));

  Device_to_String := concat(TO_STRING(e_device.Device_Null), sId);

ELSE
  IF (eMsgDevice >= e_Device.Process)
  THEN
    nId := eMsgDevice MOD e_Device.Process;
    sId := concat(sId, TO_STRING(nId));
 
    Device_to_String := concat(TO_STRING(e_Device.Process), sId);

  ELSIF (eMsgDevice >= e_Device.Data)
  THEN
    nId := eMsgDevice MOD e_Device.Data;
    sId := concat(sId, TO_STRING(nId));
 
    Device_to_String := concat(TO_STRING(e_device.Data), sId);

  ELSIF (eMsgDevice >= e_device.XfcAxis)
  THEN
    nId := eMsgDevice MOD e_device.XfcAxis;
    sId := concat(sId, TO_STRING(nId));
 
    Device_to_String := concat(TO_STRING(e_device.XfcAxis), sId);

  ELSIF (eMsgDevice >= e_device.Axis)
  THEN
    nId := eMsgDevice MOD e_device.Axis;
    sId := concat(sId, TO_STRING(nId));
 
    Device_to_String := concat(TO_STRING(e_device.Axis), sId);

  ELSIF (eMsgDevice >= e_device.NciChannelCtrl)
  THEN
    nId := eMsgDevice MOD e_device.NciChannelCtrl;
    sId := concat(sId, TO_STRING(nId));
 
    Device_to_String := concat(TO_STRING(e_device.NciChannelCtrl), sId);

  ELSIF (eMsgDevice >= e_device.NciChannel)
  THEN
    nId := eMsgDevice MOD e_device.NciChannel;
    sId := concat(sId, TO_STRING(nId));
 
    Device_to_String := concat(TO_STRING(e_device.NciChannel), sId);

  ELSIF (eMsgDevice >= e_Device.Camming)
  THEN
    nId := eMsgDevice MOD e_Device.Camming;
    sId := concat(sId, TO_STRING(nId));
 
    Device_to_String := concat(TO_STRING(e_device.Camming), sId);

  ELSIF (eMsgDevice >= e_Device.XtsStation)
  THEN
    nId := eMsgDevice MOD e_Device.XtsStation;
    sId := concat(sId, TO_STRING(nId));
 
    Device_to_String := concat(TO_STRING(e_device.XtsStation), sId);

  ELSIF (eMsgDevice >= e_Device.XfcTouchProbe)
  THEN
    nId := eMsgDevice MOD e_Device.XfcTouchProbe;
    sId := concat(sId, TO_STRING(nId));
 
    Device_to_String := concat(TO_STRING(e_device.XfcTouchProbe), sId);

  ELSIF (eMsgDevice >= e_Device.XfcTriggerBox)
  THEN
    nId := eMsgDevice MOD e_Device.XfcTriggerBox;
    sId := concat(sId, TO_STRING(nId));
 
    Device_to_String := concat(TO_STRING(e_device.XfcTriggerBox), sId);

  ELSIF (eMsgDevice >= e_Device.XtsTransportUnit)
  THEN
    nId := eMsgDevice MOD e_Device.XtsTransportUnit;
    sId := concat(sId, TO_STRING(nId));
 
    Device_to_String := concat(TO_STRING(e_device.XtsTransportUnit), sId);

  ELSIF (eMsgDevice >= e_Device.MoverCtrl)
  THEN
    nId := eMsgDevice MOD e_Device.MoverCtrl;
    sId := concat(sId, TO_STRING(nId));
 
    Device_to_String := concat(TO_STRING(e_device.MoverCtrl), sId);

  ELSIF (eMsgDevice >= e_Device.Mover)
  THEN
    nId := eMsgDevice MOD e_Device.Mover;
    sId := concat(sId, TO_STRING(nId));
 
    Device_to_String := concat(TO_STRING(e_device.Mover), sId);

  ELSIF (eMsgDevice >= e_Device.XpuCtrl)
  THEN
    nId := eMsgDevice MOD e_Device.XpuCtrl;
    sId := concat(sId, TO_STRING(nId));
 
    Device_to_String := concat(TO_STRING(e_device.XpuCtrl), sId);

  ELSIF (eMsgDevice >= e_Device.Xpu)
  THEN
    nId := eMsgDevice MOD e_Device.Xpu;
    sId := concat(sId, TO_STRING(nId));
 
    Device_to_String := concat(TO_STRING(e_device.Xpu), sId);

  ELSIF (eMsgDevice >= e_Device.CaGroup)
  THEN
    nId := eMsgDevice MOD e_Device.CaGroup;
    sId := concat(sId, TO_STRING(nId));
 
    Device_to_String := concat(TO_STRING(e_device.CaGroup), sId);

  ELSIF (eMsgDevice >= e_Device.General)
  THEN
    nId := eMsgDevice MOD e_Device.General;
    sId := concat(sId, TO_STRING(nId));
 
    Device_to_String := concat(TO_STRING(e_device.General), sId);

  ELSE
    Device_to_String := TO_STRING(eMsgDevice);
  END_IF
END_IF
END_METHOD

METHOD FolderDate : STRING
VAR_INPUT
	pLocalTime		: POINTER TO DT;
END_VAR
VAR
	sTmp					: STRING;
END_VAR
IF NOT (pLocalTime <> 0)
THEN
	FolderDate := 'NULL';
	RETURN;
END_IF

sTmp := DT_TO_STRING(pLocalTime^);

// cut off #dt literal
sTmp := right(sTmp, len(sTmp)-3);

sTmp := replace(sTmp, '_', 1, 5);
sTmp := replace(sTmp, '_', 1, 8);

sTmp := left(sTmp,10);	// year_month_day

FolderDate := sTmp;
END_METHOD

METHOD StringLen : UINT // 	string length for len > 255
VAR_INPUT
  pInString		: POINTER TO STRING(STR_LEN);
END_VAR
VAR
	Counter			: UINT;
	pInWork			: POINTER TO BYTE;
END_VAR
pInWork := pInString;
Counter := 0;

WHILE (pInWork^ <> 0) AND
			(Counter < STR_LEN)
DO
	Counter := Counter + 1;
	pInWork := pInWork + 1;
END_WHILE

StringLen := Counter;
END_METHOD

METHOD WriteData  : BOOL
VAR_INPUT
  bExecute        : BOOL;
END_VAR
VAR
END_VAR

IF NOT bExecute
THEN
  bBusyWrite                := FALSE;
	nStateWrite               := 0;
END_IF

CASE nStateWrite OF

	0:
		fbFileOpen.bExecute		  := FALSE;
		fbFileWrite.bExecute	  := FALSE;
		fbFileClose.bExecute	  := FALSE;

		IF bExecute
		THEN
			bBusyWrite            := TRUE;
			nStateWrite           := 10;
		END_IF

	10:
		fbFileOpen.bExecute     := TRUE;
		IF fbFileOpen.bBusy
		THEN
			nStateWrite           := 20;
		END_IF

	20:
		IF NOT fbFileOpen.bBusy
		THEN
			fbFileOpen.bExecute   := FALSE;
			fbFileWrite.bExecute  := TRUE;
			nStateWrite           := 30;
		END_IF

	30:
		IF fbFileWrite.bBusy
		THEN
			nStateWrite           := 40;
		END_IF

	40:
		IF NOT fbFileWrite.bBusy
		THEN
			fbFileWrite.bExecute  := FALSE;
			fbFileClose.bExecute  := TRUE;
			nStateWrite           := 50;
		END_IF

	50:
		IF fbFileClose.bBusy
		THEN
			nStateWrite           := 60;
		END_IF

	60:
		IF NOT fbFileClose.bBusy
		THEN
			fbFileClose.bExecute  := FALSE;
			nStateWrite 		      := 100;
		END_IF
	
	100:
    WriteData               := TRUE;
END_CASE


fbFileOpen(
	sNetId:= , 
	sPathName:= sFileName, 
	nMode:= FOPEN_MODEAPPEND, 
	ePath:= PATH_GENERIC, 
	bExecute:= , 
	tTimeout:= T#10S, 
	bBusy=> , 
	bError=> , 
	nErrId=> , 
	hFile=> );

fbFileWrite(
	sNetId:= , 
	hFile:= fbFileOpen.hFile, 
	pWriteBuff:= ADR(sWriteData), 
	cbWriteLen:= StringLen(ADR(sWriteData)), 
	bExecute:= , 
	tTimeout:= T#10S, 
	bBusy=> , 
	bError=> , 
	nErrId=> nErrorWrite, 
	cbWrite=> );

fbFileClose(
	sNetId:= , 
	hFile:= fbFileOpen.hFile, 
	bExecute:= , 
	tTimeout:= T#10S, 
	bBusy=> , 
	bError=> , 
	nErrId=> );

bErrorWrite := fbFileOpen.bError OR fbFileWrite.bError;
END_METHOD

END_PROGRAM

// ---- APPLICATION/MAIN_APP.TcPOU
//---------------------------------------------------------------------------------------------------------------
//
//  HAUD 2024.10.02
//
//  - APPLICATION
//    - explicit simple example PRG for setting up GearInPosCa application
//      - works dirEctly on GVL_XTS namespace Ctrl/State structs
//      - no error handling, reset application from start
//
//  - Application controls:
//    - XtsTransport
//      - GVL_XTS.TransportCtrl
//      - GVL_XTS.TransportState
//
//    - Xts Movers
//      - GVL_XTS.MoverCtrl
//      - GVL_XTS.MoverState
//      - GVL_XTS.MoverInfo
//      - GVL_XTS.MoveData
//      - GVL_XTS.GearData
//
//  - Application
//    - GearInPosCa example
//      - gear in to conveyer belt 
//
//---------------------------------------------------------------------------------------------------------------
// This SOFTWARE is provided as an Exemple by THE PROVIDER "as is" and "with all faults." THE PROVIDER makes no 
// representations or warranties of any kind concerning the safety, suitability, lack of viruses, inaccuracies, 
// typographical errors, or other harmful components of this SOFTWARE. There are inherent dangers in the use of 
// any software, and you are solely responsible for determining whether this SOFTWARE is compatible with your 
// equipment and other software installed on your equipment. You are also solely responsible for the protection 
// of your equipment and backup of your data, and THE PROVIDER will not be liable for any damages you may suffer 
// in connection with using, modifying, or distributing this SOFTWARE.
//---------------------------------------------------------------------------------------------------------------
PROGRAM MAIN_APP
VAR
  eInit         : E_PROGRESS;
  bStart        : BOOL;   // XtsTransport is initialized, CAGroup is built, All movers are enabled, XtsStations are cleared, XtsTransport base position for all movers is commanded, XtsStations are handshaked with timer
  bReset        : BOOL;   // All Xts Stations are cleared, requires new start

  nState        : UINT;   // state var for application
END_VAR



//-----------------------------------------------------------------------------
// wait for initialization to be complete before work may start
//-----------------------------------------------------------------------------
IF NOT (Main.eInit = E_PROGRESS.PROGRESS_DONE)
THEN
  eInit                               := E_PROGRESS.PROGRESS_INIT;
  bReset                              := FALSE;
  bStart                              := FALSE;
  nState                              := 0;
  RETURN;
END_IF
//-----------------------------------------------------------------------------
// fetch reset anytime
//-----------------------------------------------------------------------------
IF bReset
THEN
  bReset                              := FALSE;
  bStart                              := FALSE;
  nState                              := 9000;  // states for clearing XtsTransport
END_IF


CASE nState 
OF
  0:                                  // first PLC cycle
    nState                            := 1;

  1:
    // do other init stuff here
    eInit                             := E_PROGRESS.PROGRESS_DONE;
    nState                            := 10;

  10:                                 // starts from here
    IF bStart
    THEN
      nState                          := 100; // let's go
    END_IF
    
  100:                                // clear interface
    GVL_XTS.XtsTransportCtrl.Cmd      := E_XTS_TRANSPORT_CTRL.CMD_NULL;
    nState                            := 110;

  110:                                // check initialization of XtsTransport, wait for either MoverDetection being valid or OperationMode.Simulation
    IF (GVL_XTS.XtsTransportState.XpuInfo.IdDetectionValid) OR
       (GVL_XTS.XtsTransportState.XpuInfo.OperationMode = OperationMode.Simulation)
    THEN
      // now XtsTransport is initialized, cyclic plausibility checks on Xpu are active
      nState                          := 120;
    END_IF

  120:                                // clear group for defined start situation
    GVL_XTS.XtsTransportCtrl.Cmd      := E_XTS_TRANSPORT_CTRL.CMD_GROUP_CLEAR;

    IF (GVL_XTS.XtsTransportState.State = E_XTS_TRANSPORT_STATE.TRANSPORT_GROUP_CLEAR + E_PROGRESS.PROGRESS_DONE)
    THEN
      // CA Group is now in defined error free state
      nState                          := 130;
    END_IF

  130:                                // build Collision Avoidance group with all movers
    GVL_XTS.XtsTransportCtrl.Cmd      := E_XTS_TRANSPORT_CTRL.CMD_GROUP_BUILD;

    IF (GVL_XTS.XtsTransportState.State = E_XTS_TRANSPORT_STATE.TRANSPORT_GROUP_BUILD + E_PROGRESS.PROGRESS_DONE)
    THEN
      // CA Group contains all movers now
      // GVL_XTS.XtsTransportState.GroupInfo.AxisCount = MAX_MOVER
      nState                          := 140;
      GEAR_IN_POS_CA.bEnable          := FALSE;
      GEAR_IN_POS_CA.bReset           := FALSE;
    END_IF

  140:                                // enable CA Group
    GVL_XTS.XtsTransportCtrl.Cmd      := E_XTS_TRANSPORT_CTRL.CMD_GROUP_ENABLE;

    IF (GVL_XTS.XtsTransportState.State = E_XTS_TRANSPORT_STATE.TRANSPORT_GROUP_ENABLE + E_PROGRESS.PROGRESS_DONE)
    THEN
      // GVL_XTS.XtsTransportState.GroupInfo.CaGroupState = mcGroupStateNotReady
      nState                          := 150;
      GEAR_IN_POS_CA.bReset           := TRUE;
    END_IF

  150:                                // enable all movers
    GVL_XTS.XtsTransportCtrl.Cmd      := E_XTS_TRANSPORT_CTRL.CMD_MOVER_ENABLE;

    IF (GVL_XTS.XtsTransportState.State = E_XTS_TRANSPORT_STATE.TRANSPORT_MOVER_ENABLE + E_PROGRESS.PROGRESS_DONE)
    THEN
      // GVL_XTS.XtsTransportState.GroupInfo.CaGroupState = mcGroupStateStandby
      nState                          := 160;
      GEAR_IN_POS_CA.bReset           := FALSE;
    END_IF

  160:                                // command all movers to startup position
    GVL_XTS.XtsTransportCtrl.Cmd      := E_XTS_TRANSPORT_CTRL.CMD_TRANSPORT_START;

    IF (GVL_XTS.XtsTransportState.State = E_XTS_TRANSPORT_STATE.TRANSPORT_START + E_PROGRESS.PROGRESS_DONE)
    THEN
      // all movers are now waiting at GVL_XTS.StationStart.rPosWait
      nState                          := 1000; // go to wait state, activate GearInPos program
      // enable gear in pos sequence now the movers are ready
      GEAR_IN_POS_CA.bEnable          := TRUE;
    END_IF


  9000:
    // reset sequence trigger starts here
    GEAR_IN_POS_CA.bEnable            := FALSE;
    GVL_XTS.XtsTransportCtrl.Cmd      := E_XTS_TRANSPORT_CTRL.CMD_NULL;
    nState                            := 9005;

    GVL_APPLICATION.MasterHalt(
                        Axis          := GVL_APPLICATION.MasterAxis, 
                        Execute       := FALSE, 
                        Deceleration  :=  12500.0, 
                        Jerk          := 100000.0, 
                        BufferMode    := Tc2_MC2.MC_Aborting, 
                        Options:= , 
                        Done=> , 
                        Busy=> , 
                        Active=> , 
                        CommandAborted=> , 
                        Error=> , 
                        ErrorID=> );

  9005:
    GVL_APPLICATION.MasterHalt(
                        Axis          := GVL_APPLICATION.MasterAxis, 
                        Execute       := TRUE);

    IF (GVL_APPLICATION.MasterAxis.Status.NotMoving)
    THEN
      nState                          := 9010;

      GVL_APPLICATION.MasterHalt(
                          Axis        := GVL_APPLICATION.MasterAxis, 
                          Execute     := FALSE);

      GVL_APPLICATION.MasterPower(
                  Axis                := GVL_APPLICATION.MasterAxis, 
                  Enable              := FALSE);
    END_IF

  9010:                               // halt all movers and clear group
    GVL_XTS.XtsTransportCtrl.Cmd      := E_XTS_TRANSPORT_CTRL.CMD_GROUP_CLEAR;

    IF (GVL_XTS.XtsTransportState.State = E_XTS_TRANSPORT_STATE.TRANSPORT_GROUP_CLEAR + E_PROGRESS.PROGRESS_DONE)
    THEN
      // CA group cleared and mover in standstill
      nState                          := 9100;
    END_IF

  9100:                               // switch off movers
    GVL_XTS.XtsTransportCtrl.Cmd      := E_XTS_TRANSPORT_CTRL.CMD_MOVER_DISABLE;

    IF (GVL_XTS.XtsTransportState.State = E_XTS_TRANSPORT_STATE.TRANSPORT_MOVER_DISABLE + E_PROGRESS.PROGRESS_ERROR)
    THEN
      nState                          := 9010;
    ELSIF (GVL_XTS.XtsTransportState.State = E_XTS_TRANSPORT_STATE.TRANSPORT_MOVER_DISABLE + E_PROGRESS.PROGRESS_DONE)
    THEN
      nState                          := 10;
    END_IF

END_CASE

GVL_APPLICATION.MasterAxis(); // update master axis

GEAR_IN_POS_CA();             // gear in pos sequence

END_PROGRAM

// ---- APPLICATION/GEAR_IN_POS_CA.TcPOU
//---------------------------------------------------------------------------------------------------------------
//
//  HAUD 2024.10.02
//
//  - simple program for GearInPosCa of mover and conveyer belt (MasterAxis)
//    - mover is geared in
//    - sync distance is checked
//    - mover is sent to target position
//---------------------------------------------------------------------------------------------------------------
PROGRAM GEAR_IN_POS_CA
VAR_INPUT
  bReset                : BOOL;
  bEnable               : BOOL;
END_VAR
VAR_OUTPUT
  bError                : BOOL;
END_VAR
VAR
  nErrorId              : UDINT;

  // this example checks the sync distance of the conveyer
  rDiffPositionConveyer, 
  rStartPositionConveyer,
  rTargetPositionMover  : LREAL;

  rSyncDistance         : LREAL;
  rSyncDistanceConveyer : LREAL := 225.0;

  nState                : UINT;
  nMover                : UINT;
  rtrigReset            : Tc2_Standard.R_TRIG;
END_VAR

rtrigReset(CLK:= bReset);
IF rtrigReset.Q
THEN
  nState                       := 0;
  FOR nMover := 1 TO MAX_MOVER
  DO
    GVL_XTS.MoverCtrl[nMover].Cmd      := E_MOVER_CTRL.MOVER_NULL;
  END_FOR
END_IF





CASE nState OF
  0:
    IF bEnable AND NOT bReset
    THEN
      bError                        := FALSE;
      nErrorId                      := 0;
      nMover                        := 1;
      nState                        := 10;
    END_IF

  10:
    nState                          := 11;
    GVL_APPLICATION.MasterReset(
                      Axis          := GVL_APPLICATION.MasterAxis, 
                      Execute       := FALSE, 
                      Done=> , 
                      Busy=> , 
                      Error=> , 
                      ErrorID=> );

  11:
    GVL_APPLICATION.MasterReset(
                      Axis          := GVL_APPLICATION.MasterAxis, 
                      Execute       := TRUE);

    IF (GVL_APPLICATION.MasterReset.Done)
    THEN
      nState                        := 12;
    END_IF

  12:
    nState                          := 13;
    GVL_APPLICATION.MasterReset(
                      Axis          := GVL_APPLICATION.MasterAxis, 
                      Execute       := FALSE);

  13:
    GVL_APPLICATION.MasterPower(
                Axis                := GVL_APPLICATION.MasterAxis, 
                Enable              := TRUE, 
                Enable_Positive     := TRUE, 
                Enable_Negative     := TRUE, 
                Override            := GVL_APPLICATION.MoveData.rOverride, 
                BufferMode:= , 
                Options:= , 
                Status=> , 
                Busy=> , 
                Error=> , 
                ErrorID=> );

    IF NOT (GVL_APPLICATION.MasterPower.Error)
    THEN
      IF (GVL_APPLICATION.MasterAxis.Status.ControlLoopClosed)
      THEN
        nState                      := 14;
      END_IF
    ELSE
      nState                        := 9000;
      nErrorId                      := GVL_APPLICATION.MasterPower.ErrorID;
    END_IF

  14:
    nState                          := 15;

    // READ THIS:
    // https://infosys.beckhoff.com/english.php?content=../content/1033/tf5410_tc3_collision_avoidance/1534969995.html&id=

    GVL_APPLICATION.MoveData.rVelo  :=  1000.0;   // dynamics for gearing procedure
    GVL_APPLICATION.MoveData.rAcc   := 12500.0;   // dynamics for gearing procedure
    GVL_APPLICATION.MoveData.rGap   :=   100.0;   // gap which has to be maintained during operations

    GVL_APPLICATION.GearData.rDeltaToMasterPos      :=  125.0;  // distance to GearIn position of master
    GVL_APPLICATION.GearData.rMasterStartDistance   :=    0.0;  // distance master has to move until gearing is started
    GVL_APPLICATION.GearData.rModuloSyncPosSlave    :=   75.0;  // Modulo Position of mover where master and mover have to be in sync
    GVL_APPLICATION.GearData.rGearNumerator         :=    1.0;  // Gearing factor

    GVL_APPLICATION.MasterMoveVelo(
                  Axis              := GVL_APPLICATION.MasterAxis, 
                  Execute           := FALSE, 
                  Velocity          :=    500.0, 
                  Acceleration      :=  12500.0, 
                  Deceleration      :=  12500.0, 
                  Jerk              := 100000.0, 
                  Direction         := Tc2_MC2.MC_Direction.MC_Positive_Direction, 
                  BufferMode        := Tc2_MC2.MC_Aborting, 
                  Options:= , 
                  InVelocity=> , 
                  Busy=> , 
                  Active=> , 
                  CommandAborted=> , 
                  Error=> , 
                  ErrorID=> );

  15:
    GVL_APPLICATION.MasterMoveVelo(
                  Axis              := GVL_APPLICATION.MasterAxis, 
                  Execute           := TRUE);

    IF (GVL_APPLICATION.MasterMoveVelo.Error)
    THEN
      nState                        := 9000;
      nErrorId                      := GVL_APPLICATION.MasterMoveVelo.ErrorID;

    ELSIF (GVL_APPLICATION.MasterMoveVelo.InVelocity)
    THEN
      nState                        := 1000;
    END_IF


  1000:
    IF bEnable
    THEN
      nState                        := 1010;
      // see method fb_Mover.GearInPosCa for how the MC_GearInPosCa is connected
      // GVL_XTS.MoverCtrl is triggering fb_MoverCtrl(fb_Mover) instance
      GVL_XTS.MoveData [nMover]     := GVL_APPLICATION.MoveData;  // feed dynamic constraints into datafield of mover
      GVL_XTS.GearData [nMover]     := GVL_APPLICATION.GearData;  // feed gearing constraints into datafield of mover

      GVL_XTS.MoverCtrl[nMover].Cmd := E_MOVER_CTRL.MOVER_GEAR_IN_POS_CA; // start gearing procedure 
    END_IF

  1010:
    IF (GVL_XTS.MoverState[nMover].State = E_MOVER_STATE.MOVER_GEAR_IN_POS_CA + E_PROGRESS.PROGRESS_ERROR)
    THEN
      nErrorId                      := GVL_XTS.MoverInfo[nMover].nErrorId;
      nState                        := 9000;

    ELSIF (GVL_XTS.MoverState[nMover].State = E_MOVER_STATE.MOVER_GEAR_IN_POS_CA + E_PROGRESS.PROGRESS_DONE)
    THEN
      // sync movement is reached, now check for SyncDistance and then send mover away
      nState                        := 1020;
      rDiffPositionConveyer         := GVL_APPLICATION.MasterAxis.NcToPlc.ActPos - rStartPositionConveyer;
      rStartPositionConveyer        := GVL_APPLICATION.MasterAxis.NcToPlc.ActPos;
      rTargetPositionMover          := GVL_XTS.MoverItf [nMover].RailLength + GVL_XTS.StationStart.rPosWait; // this example sends movers one RailLength forward to startup position 
    END_IF

  1020:
    rSyncDistance                   := GVL_APPLICATION.MasterAxis.NcToPlc.ActPos - rStartPositionConveyer;
    IF (rSyncDistance > rSyncDistanceConveyer)
    THEN
      // sync distance is reached, now send mover away
      nState                              := 1030;
      GVL_XTS.MoveData [nMover].rPos      := rTargetPositionMover;
      GVL_XTS.MoveData [nMover].rGap      := GVL_XTS.StationStart.rGap;
      GVL_XTS.MoveData [nMover].rDistance := -5.0; // mover has to move more than this distance, then E_MOVER_CTRL.MOVER_SEND_TO_POS_CA is done

      GVL_XTS.MoverCtrl[nMover].Cmd := E_MOVER_CTRL.MOVER_SEND_TO_POS_CA;
    END_IF

  1030:
    IF (GVL_XTS.MoverState[nMover].State = E_MOVER_STATE.MOVER_SEND_TO_POS_CA + E_PROGRESS.PROGRESS_ERROR)
    THEN
      nErrorId                      := GVL_XTS.MoverInfo[nMover].nErrorId;
      nState                        := 9000;

    ELSIF (GVL_XTS.MoverState[nMover].State = E_MOVER_STATE.MOVER_SEND_TO_POS_CA + E_PROGRESS.PROGRESS_DONE)
    THEN
      nState                        := 1040;
    END_IF

  1040:
    nState                          := 1000;
    IF (nMover > MAX_MOVER-1)
    THEN
      nMover                        := 1;
    ELSE
      nMover                        := nMover + 1;
    END_IF

  9000:
    bError                          := TRUE;
END_CASE

END_PROGRAM

// ---- MSG/fb_LocalTime.TcPOU
FUNCTION_BLOCK fb_LocalTime
VAR_INPUT

END_VAR
VAR_OUTPUT
  sLocalTime  : STRING;
  dtLocalTime : DT;
END_VAR
VAR
  GetSysTime    : FW_GetSystemTime;
  strFileTime   : T_FILETIME;
END_VAR

GetSysTime(dwTimeLo=> strFileTime.dwLowDateTime, dwTimeHi=> strFileTime.dwHighDateTime);

sLocalTime := SYSTEMTIME_TO_STRING( FILETIME_TO_SYSTEMTIME( strFileTime ) );
dtLocalTime := systemtime_to_dt( FILETIME_TO_SYSTEMTIME( strFileTime ) );

END_FUNCTION_BLOCK

// ---- XTS/XtsStation/fb_Station.TcPOU
//---------------------------------------------------------------------------------------------------------------
//
//  HAUD 2023.03.07
//
//  - XTS_TRANSPORT_LAYER
//
//  fb_Station
//  - handshake with extern control for mover transport through station
//
//---------------------------------------------------------------------------------------------------------------
// This SOFTWARE is provided as an Exemple by THE PROVIDER "as is" and "with all faults." THE PROVIDER makes no 
// representations or warranties of any kind concerning the safety, suitability, lack of viruses, inaccuracies, 
// typographical errors, or other harmful components of this SOFTWARE. There are inherent dangers in the use of 
// any software, and you are solely responsible for determining whether this SOFTWARE is compatible with your 
// equipment and other software installed on your equipment. You are also solely responsible for the protection 
// of your equipment and backup of your data, and THE PROVIDER will not be liable for any damages you may suffer 
// in connection with using, modifying, or distributing this SOFTWARE.
//---------------------------------------------------------------------------------------------------------------
FUNCTION_BLOCK fb_Station IMPLEMENTS I_XtsTransport_Station
VAR
  _nStationId                 : UINT;         // why is Gamora?

  _sState                     : STRING(255);  // additional output for Check()

  _eInitList                  : E_PROGRESS;   // linked list initialization progress

  _eFatalError                : E_STATION_STATE;

  // pointer to all stations
  _stCtrl                     : REFERENCE TO ARRAY[1..MAX_STATION]  OF ST_STATION_CTRL;
  _stState                    : REFERENCE TO ARRAY[1..MAX_STATION]  OF ST_STATION_STATE;

  // local copy of command
  _eCmd,
  _eCmdOld                    : E_STATION_CTRL;

  _ItfStation                 : REFERENCE TO ARRAY[1..MAX_STATION]  OF I_Station_LinkedList;  // access to all stations lists
  _ItfMover                   : REFERENCE TO ARRAY[1..MAX_MOVER]    OF I_XtsTransport_Mover;  // access to mover methods

  // station related data
  _rMoverOffset               : REFERENCE TO ARRAY[1..MAX_STATION]  OF T_NEST_OFFSET;         // static offsets for station
  _stParameter                : REFERENCE TO ARRAY[1..MAX_STATION]  OF ST_STATION_PARAMETER;  // station parameter (where, how fast, how many stops)

  // mover axis ref for info
  _Mover                      : REFERENCE TO ARRAY[1..MAX_MOVER]    OF AXIS_REF;              // read from AXIS_REF

  // linked list result struct
  _stListEnter,
  _stListTarget,
  _stListDelete               : ST_STATION_LIST_RESULT;   // struct with result and ticket data

  _stMoverDataSend,
  _stMoverData                : ST_STATION_MOVER_DATA;    // mover ticket data

  _stInfeed,
  _stOutfeed                  : ST_MOVE_DATA;             // position and dynamic constraints of movement

  // work vars
  _Result                     : E_PROGRESS;
  _eStateProgress             : E_PROGRESS;

  _nNest,
  _nMoverDetected,
  _ix                         : UINT;

  _rModActPosFetch            : LREAL;
  _stMsg                      : ST_Message;
  _eMessageLevel              : E_MessageType;
  _bMatchMessageLevel         : BOOL := TRUE;   // TRUE --> Mover in Station commands have equal message level as station
END_VAR

METHOD PRIVATE Check : BOOL
VAR_INPUT
END_VAR
IF NOT (_nStationId > 0) OR
       (_nStationId > MAX_STATION)
THEN
  _sState                     := 'invalid nStationId';
  RETURN;
END_IF

IF NOT __ISVALIDREF(_stCtrl)
THEN
  _sState                     := '_stCtrl: missing pointer';
  RETURN;
END_IF

IF NOT __ISVALIDREF(_stState)
THEN
  _sState                     := '_stState: missing pointer';
  RETURN;
END_IF

IF NOT __ISVALIDREF(_ItfStation)
THEN
  _sState                     := '_ItfStation: missing interface';
  RETURN;
END_IF

IF NOT __ISVALIDREF(_ItfMover)
THEN
  _sState                     := '_ItfMover: missing interface';
  RETURN;
END_IF

IF NOT __ISVALIDREF(_rMoverOffset)
THEN
  _sState                     := '_rMoverOffset: missing pointer';
  RETURN;
END_IF

IF NOT __ISVALIDREF(_stParameter)
THEN
  _sState                     := '_stParameter: missing pointer';
  RETURN;
END_IF

IF NOT __ISVALIDREF(_Mover)
THEN
  _sState                     := '_Mover: missing pointer';
  RETURN;
END_IF


_sState                       := 'CHECK_DONE';
Check                         := TRUE;
END_METHOD

PROPERTY Ctrl : reference to ARRAY[1..MAX_STATION] OF ST_STATION_CTRL
SET
_stCtrl ref= Ctrl;
END_SET
END_PROPERTY

METHOD Cycle
//-----------------------------------------------------------------------------
//-----------------------------------------------------------------------------
// check pointer and interface
//-----------------------------------------------------------------------------
IF NOT Check() THEN RETURN; END_IF
//-----------------------------------------------------------------------------
//-----------------------------------------------------------------------------
// set message device ID
//-----------------------------------------------------------------------------
_stMsg.eDevice                        := e_Device.XtsStation + _nStationId;
//-----------------------------------------------------------------------------
//-----------------------------------------------------------------------------
// log command change
//-----------------------------------------------------------------------------
_eCmd                                 := _stCtrl[_nStationId].eCmd;
IF (_eCmd <> _eCmdOld)
THEN
  _eCmdOld                            := _eCmd;

  _stMsg.eType                        := E_MessageType.eMessageInfo;
  _stMsg.eSubdevice                   := StationControl;
  _stMsg.iErrorNumber                 := 0;
  _stMsg.sText                        := TO_STRING(_eCmd);

  IF (_eMessageLevel > E_MessageType.eMessageWarning)
  THEN
    f_MessageSet(_stMsg);
  END_IF
END_IF
//-----------------------------------------------------------------------------
//-----------------------------------------------------------------------------
// clear station on demand
//-----------------------------------------------------------------------------
CASE _stCtrl[_nStationId].eCmd
OF
  E_STATION_CTRL.STATION_INIT:        // commanded init from cyclic interface
    _eInitList                        := Init();
    _stState[_nStationId].rMoverModPos:= 0.0;
    _stState[_nStationId].nQueue      := TO_USINT(_ItfStation[_nStationId].Count);
    RETURN;
END_CASE
//-----------------------------------------------------------------------------
//-----------------------------------------------------------------------------
// station startup and init states
//-----------------------------------------------------------------------------
CASE _stState[_nStationId].eState
OF
  E_STATION_STATE.STATION_NO_INIT:    // startup state in first PLC cycle, init linked list required
    _eInitList                        := Init();

  E_STATION_STATE.STATION_INIT:       // switch state as reserve for anything you might add here
    _stState[_nStationId].eState      := E_STATION_STATE.STATION_DISABLE;
END_CASE
//-----------------------------------------------------------------------------
//-----------------------------------------------------------------------------
//  station disabled after init 
//  wait for command to enable
//  return state after a mover has left station
//  fall back state before entry was allowed and you decided to disable
//-----------------------------------------------------------------------------
CASE _stState[_nStationId].eState
OF
  E_STATION_STATE.STATION_DISABLE:
    IF (_stCtrl[_nStationId].eCmd = E_STATION_CTRL.STATION_ENABLE)
    THEN
      _stState[_nStationId].eState    := E_STATION_STATE.STATION_ENABLE;
    END_IF


  E_STATION_STATE.STATION_ENABLE:     // enable state is detectable on the interface for one cycle only
                                      // double check commanded enable and clear work vars
    IF (_stCtrl[_nStationId].eCmd = E_STATION_CTRL.STATION_ENABLE)
    THEN
      memset(ADR(_stListEnter),    0, SIZEOF(_stListEnter));

      _eStateProgress                 := E_PROGRESS.PROGRESS_INIT;  // substate for procedures within one state
      _stState[_nStationId].eState    := E_STATION_STATE.STATION_DETECT_MOVER;  // switch to mover detection

      IF (_eMessageLevel = E_MessageType.eMessageVerbose)
      THEN
        _stMsg.eType                  := _eMessageLevel;
        LogState(_stMsg.eType);
      END_IF
    END_IF
END_CASE
//-----------------------------------------------------------------------------
//-----------------------------------------------------------------------------
//  detection state
//   - wait until mover data is entered into list
//
//  check for disable command; fall back to disabled state
//  check linked list for new entry; proceed to request infeed of mover
//-----------------------------------------------------------------------------
CASE _stState[_nStationId].eState
OF
  E_STATION_STATE.STATION_DETECT_MOVER:// wait state for mover detection
    CASE _eStateProgress
    OF
      E_PROGRESS.PROGRESS_INIT:
        IF (_stCtrl[_nStationId].eCmd = E_STATION_CTRL.STATION_DISABLE) // check for commanded disable
        THEN
          IF (_eMessageLevel = E_MessageType.eMessageVerbose)
          THEN
            _stMsg.eType              := E_MessageType.eMessageVerbose;
            _stMsg.eSubdevice         := Stationstate;
            _stMsg.iErrorNumber       := _stState[_nStationId].nMoverId;
            _stMsg.sText              := concat(TO_STRING(_stState[_nStationId].eState), ': ');
            _stMsg.sText              := concat(_stMsg.sText, TO_STRING(E_STATION_STATE.STATION_DISABLE));
            f_MessageSet(_stMsg);
          END_IF
          _stState[_nStationId].eState      := E_STATION_STATE.STATION_DISABLE; // go back and wait, no matter the queue

        ELSIF (_ItfStation[_nStationId].Count > 0)
        THEN
          // someone entered something in my list
          _stListEnter                := _ItfStation[_nStationId].GetHead();
          _eStateProgress             := E_PROGRESS.PROGRESS_BUSY;  // go check list result data

          IF (_eMessageLevel > E_MessageType.eMessageWarning)
          THEN
            _stMsg.eType              := E_MessageType.eMessageInfo;
            _stMsg.eSubdevice         := Stationstate;
            _stMsg.iErrorNumber       := _stState[_nStationId].nMoverId;
            _stMsg.sText              := concat(TO_STRING(_stState[_nStationId].eState), ': ');
            _stMsg.sText              := concat(_stMsg.sText, TO_STRING(_eStateProgress));
            f_MessageSet(_stMsg);
          END_IF
        END_IF
    END_CASE
    CASE _eStateProgress
    OF
      E_PROGRESS.PROGRESS_BUSY:
        IF (_stListEnter.wState = 0)  // GetHead() without error
        THEN
          _stMsg.eType                := E_MessageType.eMessageVerbose;
          _stMsg.eSubdevice           := e_Subdevice.StationGetHead;
          _stMsg.iErrorNumber         := _stListEnter.stData.nMoverId;
          _stMsg.sText                := '';
          IF (_eMessageLevel = E_MessageType.eMessageVerbose)
          THEN
            f_MessageSet(_stMsg);
          END_IF

          // list is giving head as result
          _stMoverData                := _stListEnter.stData; // copy ticket from list result
          _eStateProgress             := E_PROGRESS.PROGRESS_PREPARE; // go check plausibility of ticket

          IF (_eMessageLevel = E_MessageType.eMessageVerbose)
          THEN
            _stMsg.eType              := E_MessageType.eMessageVerbose;
            _stMsg.eSubdevice         := Stationstate;
            _stMsg.iErrorNumber       := _stState[_nStationId].nMoverId;
            _stMsg.sText              := concat(TO_STRING(_stState[_nStationId].eState), ': ');
            _stMsg.sText              := concat(_stMsg.sText, TO_STRING(_eStateProgress));
            f_MessageSet(_stMsg);
          END_IF
        ELSE
          // the thing that must not be: GetHead() with error
          _stState[_nStationId].eState      := E_STATION_STATE.STATION_ERROR_LIST_GET_HEAD_FAULT; // fatal error

          _stMsg.eType                      := E_MessageType.eMessageError;
          LogState(_stMsg.eType);
        END_IF
    END_CASE
    CASE _eStateProgress
    OF
      E_PROGRESS.PROGRESS_PREPARE:    // check ticket (list entry)
        // check target assignement
        IF NOT (_stMoverData.nTargetStation = _nStationId)
        THEN
          // for whom the mover calls
          // wrong address, right mover?
          _stState[_nStationId].eState      := E_STATION_STATE.STATION_ERROR_LIST_STATION_ID_WRONG; // ctrl has to fix this, go tell ctrl

          _stMsg.eType                      := E_MessageType.eMessageWarning;
          LogState(_stMsg.eType);
        ELSE
          // it's a me
          _nMoverDetected                   := _stMoverData.nMoverId;

          IF (_nMoverDetected < 1) OR
             (_nMoverDetected > MAX_MOVER)
          THEN
            // out of range the mover must not be
            _stState[_nStationId].eState    := E_STATION_STATE.STATION_ERROR_LIST_MOVER_ID_INVALID; // fatal error

            _stMsg.eType                    := E_MessageType.eMessageError;
            LogState(_stMsg.eType);
          ELSE
            memset(ADR(_stListDelete),   0, SIZEOF(_stListDelete)); // clear work var
            _eStateProgress                 := E_PROGRESS.PROGRESS_INIT; // clear progress for next station state

            // prepare station state for new mover
            _stState[_nStationId].nMoverId  := TO_USINT(_nMoverDetected); // who is waiting to enter
            _stState[_nStationId].nMask     := _stMoverData.nMask;        // how many stops have to be made
            _stState[_nStationId].eState    := E_STATION_STATE.STATION_MOVER_ENTER; // go ask for permission to enter

            IF (_eMessageLevel > E_MessageType.eMessageWarning)
            THEN
              _stMsg.eType            := E_MessageType.eMessageInfo;
              _stMsg.eSubdevice       := Stationstate;
              _stMsg.iErrorNumber     := _stState[_nStationId].nMoverId;
              _stMsg.sText            := concat(TO_STRING(_stState[_nStationId].eState), ': ');
              _stMsg.sText            := concat(_stMsg.sText, TO_STRING(_eStateProgress));
              f_MessageSet(_stMsg);
            END_IF
          END_IF
        END_IF
    END_CASE
END_CASE
//-----------------------------------------------------------------------------
//-----------------------------------------------------------------------------
// enter into station state
//  last check for disable command; fall back to disabled state
//  check for command to enter; prepare moverment, start movement
//  check for command to skip; prepare movement, switch to outfeed state
//-----------------------------------------------------------------------------
CASE _stState[_nStationId].eState
OF
  E_STATION_STATE.STATION_MOVER_ENTER:          // requesting permission for mover to enter station
    CASE _eStateProgress
    OF
      E_PROGRESS.PROGRESS_INIT:

        CASE _stCtrl[_nStationId].eCmd
        OF
          E_STATION_CTRL.STATION_DISABLE:       // control decided to disable, mover will wait
            _stState[_nStationId].eState    := E_STATION_STATE.STATION_DISABLE;

            IF (_eMessageLevel = E_MessageType.eMessageVerbose)
            THEN
              _stMsg.eType                  := _eMessageLevel;
              LogState(_stMsg.eType);
            END_IF

          E_STATION_CTRL.STATION_MOVER_ENTER:   // control decided to let mover enter
            _nNest                    := 1;     // default nest/PosStop[1]
            _eStateProgress           := E_PROGRESS.PROGRESS_BUSY;

            IF (_eMessageLevel = E_MessageType.eMessageVerbose)
            THEN
              _stMsg.eType            := E_MessageType.eMessageVerbose;
              _stMsg.eSubdevice       := Stationstate;
              _stMsg.iErrorNumber     := _stState[_nStationId].nMoverId;
              _stMsg.sText            := concat(TO_STRING(_stState[_nStationId].eState), ': ');
              _stMsg.sText            := concat(_stMsg.sText, TO_STRING(_eStateProgress));
              f_MessageSet(_stMsg);
            END_IF

            FOR _ix := 1 TO _stParameter[_nStationId].nConfiguredStopCount
            DO
              IF GetBitWord(_stMoverData.nMask, _ix-1)
              THEN
                _nNest                := _ix;
                EXIT;
              END_IF
            END_FOR

          E_STATION_CTRL.STATION_MOVER_SEND:    // control decided to send mover away
            _stOutfeed.rDistance          := _stParameter[_nStationId].rReleaseDistance;
            _stState[_nStationId].eState  := E_STATION_STATE.STATION_MOVER_OUT;

            IF (_eMessageLevel = E_MessageType.eMessageVerbose)
            THEN
              _stMsg.eType                := _eMessageLevel;
              LogState(_stMsg.eType);
            END_IF
        END_CASE
    END_CASE
    CASE _eStateProgress
    OF
      E_PROGRESS.PROGRESS_BUSY:
        MoveData();                   // prepare movement into station

        // check if infeed movement has to cross modulo turn
        _rModActPosFetch              := _Mover[_stMoverData.nMoverId].NcToPlc.ModuloActPos;

        IF (_rModActPosFetch > _stInfeed.rPos + _stParameter[_nStationId].rReleaseDistance)
        THEN
          _stInfeed.rPos              := _stInfeed.rPos + TO_REAL(_ItfMover[_stMoverData.nMoverId].RailLength);
        END_IF

        _stState[_nStationId].eState  := E_STATION_STATE.STATION_MOVER_IN_TARGET;

        IF (_eMessageLevel = E_MessageType.eMessageVerbose)
        THEN
          _stMsg.eType                := _eMessageLevel;
          LogState(_stMsg.eType);
        END_IF
    END_CASE
END_CASE
//-----------------------------------------------------------------------------
//-----------------------------------------------------------------------------
// move into station state
//  wait for movement to be done; mover in position and standstill
//    switch state to process handshake
//-----------------------------------------------------------------------------
CASE _stState[_nStationId].eState
OF
  E_STATION_STATE.STATION_MOVER_IN_TARGET:
    _ItfMover[_stMoverData.nMoverId].MessageLevel := SEL(_bMatchMessageLevel, E_MessageType.eMessageError, _eMessageLevel);

    _Result := _ItfMover[_stState[_nStationId].nMoverId].MoveToPosCa(TRUE, _stInfeed);

    IF (_Result = E_PROGRESS.PROGRESS_DONE)
    THEN
      // mother! has arrived
      _ItfMover[_stState[_nStationId].nMoverId].MoveToPosCa(FALSE, _stInfeed);
      _stState[_nStationId].eState    := E_STATION_STATE.STATION_PROCESS_START;

      IF (_eMessageLevel > E_MessageType.eMessageWarning)
      THEN
        _stMsg.eType                  := E_MessageType.eMessageInfo;
        LogState(_stMsg.eType);
      END_IF
    ELSE
      IF (_Result = E_PROGRESS.PROGRESS_ERROR)
      THEN
        _ItfMover[_stState[_nStationId].nMoverId].MoveToPosCa(FALSE, _stInfeed);
        _stState[_nStationId].eState  := E_STATION_STATE.STATION_ERROR_INFEED_ERROR; // ctrl has to fix this, go tell ctrl

        _stMsg.eType                  := E_MessageType.eMessageError;
        LogState(_stMsg.eType);
      END_IF 
    END_IF
END_CASE
//-----------------------------------------------------------------------------
//-----------------------------------------------------------------------------
// process handshake state
//  clear bit in mask
//-----------------------------------------------------------------------------
CASE _stState[_nStationId].eState
OF
  E_STATION_STATE.STATION_PROCESS_START:
    IF (_stCtrl[_nStationId].eCmd = E_STATION_CTRL.STATION_PROCESS_START) OR  // double handshake, your choice
       (_stCtrl[_nStationId].eCmd = E_STATION_CTRL.STATION_PROCESS_DONE)      // single handshake, your choice
    THEN
      // clear bit in mask when started/done
      _stState[_nStationId].nMask     := TO_USINT(DelBitWord(TO_WORD(_stState[_nStationId].nMask), _nNest-1));
      _stState[_nStationId].eState    := E_STATION_STATE.STATION_PROCESS_DONE;

      IF (_eMessageLevel = E_MessageType.eMessageVerbose)
      THEN
        _stMsg.eType                  := _eMessageLevel;
        LogState(_stMsg.eType);
      END_IF
    END_IF
END_CASE
//-----------------------------------------------------------------------------
//-----------------------------------------------------------------------------
CASE _stState[_nStationId].eState
OF
  E_STATION_STATE.STATION_PROCESS_DONE:
    IF (_stCtrl[_nStationId].eCmd = E_STATION_CTRL.STATION_PROCESS_DONE)
    THEN
      _stState[_nStationId].eState    := E_STATION_STATE.STATION_CHECK;
    END_IF
END_CASE
//-----------------------------------------------------------------------------
//-----------------------------------------------------------------------------
// check state if the mover has to move to another nest or must leave station
//-----------------------------------------------------------------------------
CASE _stState[_nStationId].eState
OF
  E_STATION_STATE.STATION_CHECK:
    IF (_stState[_nStationId].nMask = 0)
    THEN
      // mover has to leave
      _stState[_nStationId].eState    := E_STATION_STATE.STATION_MOVER_OUT;

      IF (_eMessageLevel = E_MessageType.eMessageVerbose)
      THEN
        _stMsg.eType                  := _eMessageLevel;
        LogState(_stMsg.eType);
      END_IF
    ELSE
      // _stState[_nStationId].nMask <> 0
      FOR _ix := 1 TO MAX_STATION_NEST
      DO
        IF NOT (_ix > _stParameter[_nStationId].nConfiguredStopCount)
        THEN
          IF GetBitWord(_stState[_nStationId].nMask, _ix-1)
          THEN
            // more work to do
            _stState[_nStationId].eState  := E_STATION_STATE.STATION_CHECK_NEST;
            _nNest                        := _ix; // index to move to

            IF (_eMessageLevel = E_MessageType.eMessageVerbose)
            THEN
              _stMsg.eType                := _eMessageLevel;
              LogState(_stMsg.eType);
            END_IF
            EXIT;
          END_IF
        ELSE
          IF GetBitWord(_stState[_nStationId].nMask, _ix-1)
          THEN
            // not configured, not worked
            _stMsg.eType              := E_MessageType.eMessageWarning;
            _stMsg.eSubdevice         := Stationstate;
            _stMsg.iErrorNumber       := _ix;
            _stMsg.sText              := concat(TO_STRING(_stState[_nStationId].eState), ': ');
            _stMsg.sText              := concat(_stMsg.sText, Tc2_Utilities.BYTE_TO_BINSTR(_stState[_nStationId].nMask, TO_INT(MAX_STATION_NEST)));
            IF (_eMessageLevel > E_MessageType.eMessageError)
            THEN
              f_MessageSet(_stMsg);
            END_IF

            _stState[_nStationId].nMask := TO_USINT(DelBitWord(TO_WORD(_stState[_nStationId].nMask), _ix-1));
          END_IF
        END_IF
      END_FOR
    END_IF
END_CASE
//-----------------------------------------------------------------------------
//-----------------------------------------------------------------------------
// wait state before movement to next nest has to be started
//-----------------------------------------------------------------------------
CASE _stState[_nStationId].eState
OF
  E_STATION_STATE.STATION_CHECK_NEST:
    IF (_stCtrl[_nStationId].eCmd = E_STATION_CTRL.STATION_MOVER_ENTER)
    THEN
      MoveData();
      _stState[_nStationId].eState    := E_STATION_STATE.STATION_MOVER_IN_TARGET;
  
      IF (_eMessageLevel = E_MessageType.eMessageVerbose)
      THEN
        _stMsg.eType                  := _eMessageLevel;
        LogState(_stMsg.eType);
      END_IF
    END_IF
END_CASE
//-----------------------------------------------------------------------------
//-----------------------------------------------------------------------------
// wait state for outfeed of mover
//  check ctrl data, target must be plausible, nTargetStation is what you have to set
//-----------------------------------------------------------------------------
CASE _stState[_nStationId].eState
OF
  E_STATION_STATE.STATION_MOVER_OUT:
    IF (_stCtrl[_nStationId].eCmd = E_STATION_CTRL.STATION_MOVER_OUT)
    THEN
      IF (_stCtrl[_nStationId].nTargetStation < 1) OR  
         (_stCtrl[_nStationId].nTargetStation > MAX_STATION)
      THEN
        _stState[_nStationId].eState  := E_STATION_STATE.STATION_ERROR_OUTFEED_TARGET_INVALID; // ctrl has to fix this, go tell ctrl

        _stMsg.eType                  := E_MessageType.eMessageError;
        LogState(_stMsg.eType);
      ELSE
        _stListDelete                 := _ItfStation[_nStationId].RemoveHeadValue(); // delete mover data in stations linked list


        IF (_stListDelete.wState <> 0)
        THEN
        // deleting mover in list was NOT successful
          _stState[_nStationId].eState:= E_STATION_STATE.STATION_ERROR_LIST_REMOVE_HEAD_FAULT; // fatal error

          _stMsg.eType                := E_MessageType.eMessageError;
          LogState(_stMsg.eType);

        ELSE
        // mover data successfully deleted
          _stMsg.eType                := E_MessageType.eMessageVerbose;
          _stMsg.eSubdevice           := e_Subdevice.StationRemoveHeadValue;
          _stMsg.iErrorNumber         := _stState[_nStationId].nMoverId;
          _stMsg.sText                := '';
          IF (_eMessageLevel = E_MessageType.eMessageVerbose)
          THEN
            f_MessageSet(_stMsg);
          END_IF

          memset(ADR(_stListTarget),   0, SIZEOF(_stListTarget)); // clear debug var

          // prepare movement and switch state to start movement
          MoverOut();
          _stState[_nStationId].eState  := E_STATION_STATE.STATION_MOVER_RELEASE;

          IF (_eMessageLevel > E_MessageType.eMessageWarning)
          THEN
            _stMsg.eType                := E_MessageType.eMessageInfo;
            LogState(_stMsg.eType);
          END_IF
        END_IF
      END_IF
    END_IF
END_CASE
//-----------------------------------------------------------------------------
//-----------------------------------------------------------------------------
// ckeck if mover has left the station
//  enter mover data into list of target station
//-----------------------------------------------------------------------------
CASE _stState[_nStationId].eState
OF
  E_STATION_STATE.STATION_MOVER_RELEASE:
    _ItfMover[_stMoverData.nMoverId].MessageLevel := SEL(_bMatchMessageLevel, E_MessageType.eMessageError, _eMessageLevel);

    _Result                           := _ItfMover[_stMoverDataSend.nMoverId].SendToModuloPosCa(TRUE, _stOutfeed);

    IF (_Result = E_PROGRESS.PROGRESS_DONE)
    THEN
      // add entry in target station list
      _stListTarget                   := _ItfStation[_stMoverDataSend.nTargetStation].AddTailValue(_stMoverDataSend);

      IF (_stListTarget.wState <> 0)
      THEN
      // adding mover in target list was NOT successful
        _stState[_nStationId].eState  := E_STATION_STATE.STATION_ERROR_LIST_ADD_TAIL_FAULT; // fatal error
        _stMsg.eType                  := E_MessageType.eMessageError;
        LogState(_stMsg.eType);

      ELSE
      // mover data successfully added to target station list
        IF (_eMessageLevel > E_MessageType.eMessageWarning)
        THEN
          _stMsg.eType                := E_MessageType.eMessageInfo;
          _stMsg.eSubdevice           := e_Subdevice.StationAddTail;
          _stMsg.iErrorNumber         := _stState[_nStationId].nMoverId;
          _stMsg.sText                := concat('TargetStation: ', TO_STRING(_stListTarget.stData.nTargetStation));
          f_MessageSet(_stMsg);
        END_IF
        _ItfMover[_stMoverDataSend.nMoverId].SendToModuloPosCa(FALSE, _stOutfeed);

        _stState[_nStationId].eState  := E_STATION_STATE.STATION_MOVER_GONE; // go tell ctrl that station is empty

        IF (_eMessageLevel = E_MessageType.eMessageVerbose)
        THEN
          _stMsg.eType                := _eMessageLevel;
          LogState(_stMsg.eType);
        END_IF
      END_IF
    ELSIF (_Result = E_PROGRESS.PROGRESS_ERROR)
    THEN
      _stState[_nStationId].eState    := E_STATION_STATE.STATION_ERROR_OUTFEED_ERROR; // ctrl has to fix this, go tell ctrl
      _stMsg.eType                    := E_MessageType.eMessageError;
      LogState(_stMsg.eType);
    END_IF
END_CASE
//-----------------------------------------------------------------------------
//-----------------------------------------------------------------------------
// check handshake for empty station
//  switch back station state for new mover to be able to enter
//-----------------------------------------------------------------------------
CASE _stState[_nStationId].eState
OF
  E_STATION_STATE.STATION_MOVER_GONE:

    memset(ADR(_stMoverData),  0, SIZEOF(_stMoverData));

    _stState[_nStationId].nMask       := 0;
    _stState[_nStationId].nMoverId    := 0;

    IF (_stCtrl[_nStationId].eCmd = E_STATION_CTRL.STATION_MOVER_GONE)
    THEN
      _stState[_nStationId].eState    := E_STATION_STATE.STATION_DISABLE;

      IF (_eMessageLevel = E_MessageType.eMessageVerbose)
      THEN
        _stMsg.eType                  := _eMessageLevel;
        LogState(_stMsg.eType);
      END_IF
    END_IF
END_CASE
//-----------------------------------------------------------------------------
//-----------------------------------------------------------------------------
_sState                               := TO_STRING(_stState[_nStationId].eState);
//-----------------------------------------------------------------------------
//-----------------------------------------------------------------------------
// Error handling
//-----------------------------------------------------------------------------
CASE _stState[_nStationId].eState
OF
  //---------------------------------------------------------------------------
  //---------------------------------------------------------------------------
  E_STATION_STATE.STATION_ERROR_LIST_STATION_ID_WRONG:
    IF (_stCtrl[_nStationId].eCmd = E_STATION_CTRL.STATION_MOVER_OUT)
    THEN
      _nMoverDetected                 := _stMoverData.nMoverId;

      IF (_nMoverDetected < 1) OR
         (_nMoverDetected > MAX_MOVER)
      THEN
        // this MUST NOT happen
        _stState[_nStationId].eState  := E_STATION_STATE.STATION_ERROR_LIST_MOVER_ID_INVALID; // fatal error
        _stMsg.eType                  := E_MessageType.eMessageError;
        LogState(_stMsg.eType);

      ELSE
        // not for station; send mover out
        _stState[_nStationId].eState  := E_STATION_STATE.STATION_MOVER_OUT;

        IF (_eMessageLevel > E_MessageType.eMessageError)
        THEN
          _stMsg.eType                := E_MessageType.eMessageInfo;
          LogState(_stMsg.eType);
        END_IF
      END_IF

    ELSIF (_stCtrl[_nStationId].eCmd = E_STATION_CTRL.STATION_MOVER_ENTER)
    THEN
      // override wrong TargetStationId in List; start infeed of mover

      _nMoverDetected                 := _stMoverData.nMoverId;

      IF (_nMoverDetected < 1) OR
         (_nMoverDetected > MAX_MOVER)
      THEN
        // this MUST NOT happen
        _stState[_nStationId].eState  := E_STATION_STATE.STATION_ERROR_LIST_MOVER_ID_INVALID; // fatal error

        _stMsg.eType                  := E_MessageType.eMessageError;
        LogState(_stMsg.eType);

      ELSE
        _eStateProgress               := E_PROGRESS.PROGRESS_INIT;
        _stState[_nStationId].nMoverId:= TO_USINT(_nMoverDetected);
        _stState[_nStationId].nMask   := _stMoverData.nMask;
        _stState[_nStationId].eState  := E_STATION_STATE.STATION_MOVER_ENTER;

        IF (_eMessageLevel > E_MessageType.eMessageError)
        THEN
          _stMsg.eType                := E_MessageType.eMessageInfo;
          LogState(_stMsg.eType);
        END_IF
      END_IF
    END_IF

  //---------------------------------------------------------------------------
  //---------------------------------------------------------------------------
  E_STATION_STATE.STATION_ERROR_OUTFEED_TARGET_INVALID:
    // wait here until valid target is detected
    IF NOT (_stCtrl[_nStationId].nTargetStation < 1) AND  
       NOT (_stCtrl[_nStationId].nTargetStation > MAX_STATION)
    THEN
      _stState[_nStationId].eState    := E_STATION_STATE.STATION_MOVER_OUT;

      IF (_eMessageLevel > E_MessageType.eMessageError)
      THEN
        _stMsg.eType                  := E_MessageType.eMessageInfo;
        LogState(_stMsg.eType);
      END_IF
    END_IF

  //---------------------------------------------------------------------------
  //---------------------------------------------------------------------------
  E_STATION_STATE.STATION_ERROR_INFEED_ERROR:   // must be fixed by extern by using cyclic mover control
    IF (_stCtrl[_nStationId].eCmd = E_STATION_CTRL.STATION_MOVER_ENTER_RETRY)
    THEN
      _stState[_nStationId].eState    := E_STATION_STATE.STATION_DETECT_MOVER;   // return to start and wait

      IF (_eMessageLevel > E_MessageType.eMessageError)
      THEN
        _stMsg.eType                  := E_MessageType.eMessageInfo;
        LogState(_stMsg.eType);
      END_IF
    END_IF


  //---------------------------------------------------------------------------
  //---------------------------------------------------------------------------
  E_STATION_STATE.STATION_ERROR_OUTFEED_ERROR:  // must be fixed by extern by using cyclic mover control
    IF (_stCtrl[_nStationId].eCmd = E_STATION_CTRL.STATION_MOVER_OUT_RETRY)
    THEN
      MoverOut();
      _stState[_nStationId].eState  := E_STATION_STATE.STATION_MOVER_RELEASE;

      IF (_eMessageLevel > E_MessageType.eMessageError)
      THEN
        _stMsg.eType                  := E_MessageType.eMessageInfo;
        LogState(_stMsg.eType);
      END_IF

    ELSIF (_stCtrl[_nStationId].eCmd = E_STATION_CTRL.STATION_MOVER_GONE)
    THEN
      MoverOut();

      // add entry in target station list
      _stListTarget                   := _ItfStation[_stMoverDataSend.nTargetStation].AddTailValue(_stMoverDataSend);
      IF (_stListTarget.wState <> 0)
      THEN
        _stState[_nStationId].eState  := E_STATION_STATE.STATION_ERROR_LIST_ADD_TAIL_FAULT; // fatal error
        _stMsg.eType                  := E_MessageType.eMessageError;
        LogState(_stMsg.eType);

